   STATUS[822].EXT.AckRequired := FALSE;
   STATUS[822].EXT.Maintanence := FALSE;
   STATUS[822].EXT.Operation := FALSE;
   STATUS[822].EXT.Forced := FALSE;
   STATUS[822].EXT.BIT29 := FALSE;
   STATUS[822].EXT.BIT30 := FALSE;
   STATUS[822].EXT.BIT31 := FALSE;
   STATUS[822].EXT.ModeBit1 := FALSE;
   STATUS[822].EXT.ModeBit2 := FALSE;
   STATUS[822].EXT.ModeBit3 := FALSE;
   STATUS[822].EXT.BIT19 := FALSE;
   STATUS[822].EXT.BIT20 := FALSE;
   STATUS[822].EXT.AlarmSuppressed := FALSE;
   STATUS[822].EXT.AlarmPresent := FALSE;
   STATUS[822].EXT.AlarmFailUnAck := FALSE;
   STATUS[822].Status := 0;
   STATUS[822].TimeStamp := 16#0000;
   STATUS[823].EXT.AlarmWarnUnAck := FALSE;
   STATUS[823].EXT.AckRequired := FALSE;
   STATUS[823].EXT.Maintanence := FALSE;
   STATUS[823].EXT.Operation := FALSE;
   STATUS[823].EXT.Forced := FALSE;
   STATUS[823].EXT.BIT29 := FALSE;
   STATUS[823].EXT.BIT30 := FALSE;
   STATUS[823].EXT.BIT31 := FALSE;
   STATUS[823].EXT.ModeBit1 := FALSE;
   STATUS[823].EXT.ModeBit2 := FALSE;
   STATUS[823].EXT.ModeBit3 := FALSE;
   STATUS[823].EXT.BIT19 := FALSE;
   STATUS[823].EXT.BIT20 := FALSE;
   STATUS[823].EXT.AlarmSuppressed := FALSE;
   STATUS[823].EXT.AlarmPresent := FALSE;
   STATUS[823].EXT.AlarmFailUnAck := FALSE;
   STATUS[823].Status := 0;
   STATUS[823].TimeStamp := 16#0000;
   STATUS[824].EXT.AlarmWarnUnAck := FALSE;
   STATUS[824].EXT.AckRequired := FALSE;
   STATUS[824].EXT.Maintanence := FALSE;
   STATUS[824].EXT.Operation := FALSE;
   STATUS[824].EXT.Forced := FALSE;
   STATUS[824].EXT.BIT29 := FALSE;
   STATUS[824].EXT.BIT30 := FALSE;
   STATUS[824].EXT.BIT31 := FALSE;
   STATUS[824].EXT.ModeBit1 := FALSE;
   STATUS[824].EXT.ModeBit2 := FALSE;
   STATUS[824].EXT.ModeBit3 := FALSE;
   STATUS[824].EXT.BIT19 := FALSE;
   STATUS[824].EXT.BIT20 := FALSE;
   STATUS[824].EXT.AlarmSuppressed := FALSE;
   STATUS[824].EXT.AlarmPresent := FALSE;
   STATUS[824].EXT.AlarmFailUnAck := FALSE;
   STATUS[824].Status := 0;
   STATUS[824].TimeStamp := 16#0000;
   STATUS[825].EXT.AlarmWarnUnAck := FALSE;
   STATUS[825].EXT.AckRequired := FALSE;
   STATUS[825].EXT.Maintanence := FALSE;
   STATUS[825].EXT.Operation := FALSE;
   STATUS[825].EXT.Forced := FALSE;
   STATUS[825].EXT.BIT29 := FALSE;
   STATUS[825].EXT.BIT30 := FALSE;
   STATUS[825].EXT.BIT31 := FALSE;
   STATUS[825].EXT.ModeBit1 := FALSE;
   STATUS[825].EXT.ModeBit2 := FALSE;
   STATUS[825].EXT.ModeBit3 := FALSE;
   STATUS[825].EXT.BIT19 := FALSE;
   STATUS[825].EXT.BIT20 := FALSE;
   STATUS[825].EXT.AlarmSuppressed := FALSE;
   STATUS[825].EXT.AlarmPresent := FALSE;
   STATUS[825].EXT.AlarmFailUnAck := FALSE;
   STATUS[825].Status := 0;
   STATUS[825].TimeStamp := 16#0000;
   STATUS[826].EXT.AlarmWarnUnAck := FALSE;
   STATUS[826].EXT.AckRequired := FALSE;
   STATUS[826].EXT.Maintanence := FALSE;
   STATUS[826].EXT.Operation := FALSE;
   STATUS[826].EXT.Forced := FALSE;
   STATUS[826].EXT.BIT29 := FALSE;
   STATUS[826].EXT.BIT30 := FALSE;
   STATUS[826].EXT.BIT31 := FALSE;
   STATUS[826].EXT.ModeBit1 := FALSE;
   STATUS[826].EXT.ModeBit2 := FALSE;
   STATUS[826].EXT.ModeBit3 := FALSE;
   STATUS[826].EXT.BIT19 := FALSE;
   STATUS[826].EXT.BIT20 := FALSE;
   STATUS[826].EXT.AlarmSuppressed := FALSE;
   STATUS[826].EXT.AlarmPresent := FALSE;
   STATUS[826].EXT.AlarmFailUnAck := FALSE;
   STATUS[826].Status := 0;
   STATUS[826].TimeStamp := 16#0000;
   STATUS[827].EXT.AlarmWarnUnAck := FALSE;
   STATUS[827].EXT.AckRequired := FALSE;
   STATUS[827].EXT.Maintanence := FALSE;
   STATUS[827].EXT.Operation := FALSE;
   STATUS[827].EXT.Forced := FALSE;
   STATUS[827].EXT.BIT29 := FALSE;
   STATUS[827].EXT.BIT30 := FALSE;
   STATUS[827].EXT.BIT31 := FALSE;
   STATUS[827].EXT.ModeBit1 := FALSE;
   STATUS[827].EXT.ModeBit2 := FALSE;
   STATUS[827].EXT.ModeBit3 := FALSE;
   STATUS[827].EXT.BIT19 := FALSE;
   STATUS[827].EXT.BIT20 := FALSE;
   STATUS[827].EXT.AlarmSuppressed := FALSE;
   STATUS[827].EXT.AlarmPresent := FALSE;
   STATUS[827].EXT.AlarmFailUnAck := FALSE;
   STATUS[827].Status := 0;
   STATUS[827].TimeStamp := 16#0000;
   STATUS[828].EXT.AlarmWarnUnAck := FALSE;
   STATUS[828].EXT.AckRequired := FALSE;
   STATUS[828].EXT.Maintanence := FALSE;
   STATUS[828].EXT.Operation := FALSE;
   STATUS[828].EXT.Forced := FALSE;
   STATUS[828].EXT.BIT29 := FALSE;
   STATUS[828].EXT.BIT30 := FALSE;
   STATUS[828].EXT.BIT31 := FALSE;
   STATUS[828].EXT.ModeBit1 := FALSE;
   STATUS[828].EXT.ModeBit2 := FALSE;
   STATUS[828].EXT.ModeBit3 := FALSE;
   STATUS[828].EXT.BIT19 := FALSE;
   STATUS[828].EXT.BIT20 := FALSE;
   STATUS[828].EXT.AlarmSuppressed := FALSE;
   STATUS[828].EXT.AlarmPresent := FALSE;
   STATUS[828].EXT.AlarmFailUnAck := FALSE;
   STATUS[828].Status := 0;
   STATUS[828].TimeStamp := 16#0000;
   STATUS[829].EXT.AlarmWarnUnAck := FALSE;
   STATUS[829].EXT.AckRequired := FALSE;
   STATUS[829].EXT.Maintanence := FALSE;
   STATUS[829].EXT.Operation := FALSE;
   STATUS[829].EXT.Forced := FALSE;
   STATUS[829].EXT.BIT29 := FALSE;
   STATUS[829].EXT.BIT30 := FALSE;
   STATUS[829].EXT.BIT31 := FALSE;
   STATUS[829].EXT.ModeBit1 := FALSE;
   STATUS[829].EXT.ModeBit2 := FALSE;
   STATUS[829].EXT.ModeBit3 := FALSE;
   STATUS[829].EXT.BIT19 := FALSE;
   STATUS[829].EXT.BIT20 := FALSE;
   STATUS[829].EXT.AlarmSuppressed := FALSE;
   STATUS[829].EXT.AlarmPresent := FALSE;
   STATUS[829].EXT.AlarmFailUnAck := FALSE;
   STATUS[829].Status := 0;
   STATUS[829].TimeStamp := 16#0000;
   STATUS[830].EXT.AlarmWarnUnAck := FALSE;
   STATUS[830].EXT.AckRequired := FALSE;
   STATUS[830].EXT.Maintanence := FALSE;
   STATUS[830].EXT.Operation := FALSE;
   STATUS[830].EXT.Forced := FALSE;
   STATUS[830].EXT.BIT29 := FALSE;
   STATUS[830].EXT.BIT30 := FALSE;
   STATUS[830].EXT.BIT31 := FALSE;
   STATUS[830].EXT.ModeBit1 := FALSE;
   STATUS[830].EXT.ModeBit2 := FALSE;
   STATUS[830].EXT.ModeBit3 := FALSE;
   STATUS[830].EXT.BIT19 := FALSE;
   STATUS[830].EXT.BIT20 := FALSE;
   STATUS[830].EXT.AlarmSuppressed := FALSE;
   STATUS[830].EXT.AlarmPresent := FALSE;
   STATUS[830].EXT.AlarmFailUnAck := FALSE;
   STATUS[830].Status := 0;
   STATUS[830].TimeStamp := 16#0000;
   STATUS[831].EXT.AlarmWarnUnAck := FALSE;
   STATUS[831].EXT.AckRequired := FALSE;
   STATUS[831].EXT.Maintanence := FALSE;
   STATUS[831].EXT.Operation := FALSE;
   STATUS[831].EXT.Forced := FALSE;
   STATUS[831].EXT.BIT29 := FALSE;
   STATUS[831].EXT.BIT30 := FALSE;
   STATUS[831].EXT.BIT31 := FALSE;
   STATUS[831].EXT.ModeBit1 := FALSE;
   STATUS[831].EXT.ModeBit2 := FALSE;
   STATUS[831].EXT.ModeBit3 := FALSE;
   STATUS[831].EXT.BIT19 := FALSE;
   STATUS[831].EXT.BIT20 := FALSE;
   STATUS[831].EXT.AlarmSuppressed := FALSE;
   STATUS[831].EXT.AlarmPresent := FALSE;
   STATUS[831].EXT.AlarmFailUnAck := FALSE;
   STATUS[831].Status := 0;
   STATUS[831].TimeStamp := 16#0000;
   STATUS[832].EXT.AlarmWarnUnAck := FALSE;
   STATUS[832].EXT.AckRequired := FALSE;
   STATUS[832].EXT.Maintanence := FALSE;
   STATUS[832].EXT.Operation := FALSE;
   STATUS[832].EXT.Forced := FALSE;
   STATUS[832].EXT.BIT29 := FALSE;
   STATUS[832].EXT.BIT30 := FALSE;
   STATUS[832].EXT.BIT31 := FALSE;
   STATUS[832].EXT.ModeBit1 := FALSE;
   STATUS[832].EXT.ModeBit2 := FALSE;
   STATUS[832].EXT.ModeBit3 := FALSE;
   STATUS[832].EXT.BIT19 := FALSE;
   STATUS[832].EXT.BIT20 := FALSE;
   STATUS[832].EXT.AlarmSuppressed := FALSE;
   STATUS[832].EXT.AlarmPresent := FALSE;
   STATUS[832].EXT.AlarmFailUnAck := FALSE;
   STATUS[832].Status := 0;
   STATUS[832].TimeStamp := 16#0000;
   STATUS[833].EXT.AlarmWarnUnAck := FALSE;
   STATUS[833].EXT.AckRequired := FALSE;
   STATUS[833].EXT.Maintanence := FALSE;
   STATUS[833].EXT.Operation := FALSE;
   STATUS[833].EXT.Forced := FALSE;
   STATUS[833].EXT.BIT29 := FALSE;
   STATUS[833].EXT.BIT30 := FALSE;
   STATUS[833].EXT.BIT31 := FALSE;
   STATUS[833].EXT.ModeBit1 := FALSE;
   STATUS[833].EXT.ModeBit2 := FALSE;
   STATUS[833].EXT.ModeBit3 := FALSE;
   STATUS[833].EXT.BIT19 := FALSE;
   STATUS[833].EXT.BIT20 := FALSE;
   STATUS[833].EXT.AlarmSuppressed := FALSE;
   STATUS[833].EXT.AlarmPresent := FALSE;
   STATUS[833].EXT.AlarmFailUnAck := FALSE;
   STATUS[833].Status := 0;
   STATUS[833].TimeStamp := 16#0000;
   STATUS[834].EXT.AlarmWarnUnAck := FALSE;
   STATUS[834].EXT.AckRequired := FALSE;
   STATUS[834].EXT.Maintanence := FALSE;
   STATUS[834].EXT.Operation := FALSE;
   STATUS[834].EXT.Forced := FALSE;
   STATUS[834].EXT.BIT29 := FALSE;
   STATUS[834].EXT.BIT30 := FALSE;
   STATUS[834].EXT.BIT31 := FALSE;
   STATUS[834].EXT.ModeBit1 := FALSE;
   STATUS[834].EXT.ModeBit2 := FALSE;
   STATUS[834].EXT.ModeBit3 := FALSE;
   STATUS[834].EXT.BIT19 := FALSE;
   STATUS[834].EXT.BIT20 := FALSE;
   STATUS[834].EXT.AlarmSuppressed := FALSE;
   STATUS[834].EXT.AlarmPresent := FALSE;
   STATUS[834].EXT.AlarmFailUnAck := FALSE;
   STATUS[834].Status := 0;
   STATUS[834].TimeStamp := 16#0000;
   STATUS[835].EXT.AlarmWarnUnAck := FALSE;
   STATUS[835].EXT.AckRequired := FALSE;
   STATUS[835].EXT.Maintanence := FALSE;
   STATUS[835].EXT.Operation := FALSE;
   STATUS[835].EXT.Forced := FALSE;
   STATUS[835].EXT.BIT29 := FALSE;
   STATUS[835].EXT.BIT30 := FALSE;
   STATUS[835].EXT.BIT31 := FALSE;
   STATUS[835].EXT.ModeBit1 := FALSE;
   STATUS[835].EXT.ModeBit2 := FALSE;
   STATUS[835].EXT.ModeBit3 := FALSE;
   STATUS[835].EXT.BIT19 := FALSE;
   STATUS[835].EXT.BIT20 := FALSE;
   STATUS[835].EXT.AlarmSuppressed := FALSE;
   STATUS[835].EXT.AlarmPresent := FALSE;
   STATUS[835].EXT.AlarmFailUnAck := FALSE;
   STATUS[835].Status := 0;
   STATUS[835].TimeStamp := 16#0000;
   STATUS[836].EXT.AlarmWarnUnAck := FALSE;
   STATUS[836].EXT.AckRequired := FALSE;
   STATUS[836].EXT.Maintanence := FALSE;
   STATUS[836].EXT.Operation := FALSE;
   STATUS[836].EXT.Forced := FALSE;
   STATUS[836].EXT.BIT29 := FALSE;
   STATUS[836].EXT.BIT30 := FALSE;
   STATUS[836].EXT.BIT31 := FALSE;
   STATUS[836].EXT.ModeBit1 := FALSE;
   STATUS[836].EXT.ModeBit2 := FALSE;
   STATUS[836].EXT.ModeBit3 := FALSE;
   STATUS[836].EXT.BIT19 := FALSE;
   STATUS[836].EXT.BIT20 := FALSE;
   STATUS[836].EXT.AlarmSuppressed := FALSE;
   STATUS[836].EXT.AlarmPresent := FALSE;
   STATUS[836].EXT.AlarmFailUnAck := FALSE;
   STATUS[836].Status := 0;
   STATUS[836].TimeStamp := 16#0000;
   STATUS[837].EXT.AlarmWarnUnAck := FALSE;
   STATUS[837].EXT.AckRequired := FALSE;
   STATUS[837].EXT.Maintanence := FALSE;
   STATUS[837].EXT.Operation := FALSE;
   STATUS[837].EXT.Forced := FALSE;
   STATUS[837].EXT.BIT29 := FALSE;
   STATUS[837].EXT.BIT30 := FALSE;
   STATUS[837].EXT.BIT31 := FALSE;
   STATUS[837].EXT.ModeBit1 := FALSE;
   STATUS[837].EXT.ModeBit2 := FALSE;
   STATUS[837].EXT.ModeBit3 := FALSE;
   STATUS[837].EXT.BIT19 := FALSE;
   STATUS[837].EXT.BIT20 := FALSE;
   STATUS[837].EXT.AlarmSuppressed := FALSE;
   STATUS[837].EXT.AlarmPresent := FALSE;
   STATUS[837].EXT.AlarmFailUnAck := FALSE;
   STATUS[837].Status := 0;
   STATUS[837].TimeStamp := 16#0000;
   STATUS[838].EXT.AlarmWarnUnAck := FALSE;
   STATUS[838].EXT.AckRequired := FALSE;
   STATUS[838].EXT.Maintanence := FALSE;
   STATUS[838].EXT.Operation := FALSE;
   STATUS[838].EXT.Forced := FALSE;
   STATUS[838].EXT.BIT29 := FALSE;
   STATUS[838].EXT.BIT30 := FALSE;
   STATUS[838].EXT.BIT31 := FALSE;
   STATUS[838].EXT.ModeBit1 := FALSE;
   STATUS[838].EXT.ModeBit2 := FALSE;
   STATUS[838].EXT.ModeBit3 := FALSE;
   STATUS[838].EXT.BIT19 := FALSE;
   STATUS[838].EXT.BIT20 := FALSE;
   STATUS[838].EXT.AlarmSuppressed := FALSE;
   STATUS[838].EXT.AlarmPresent := FALSE;
   STATUS[838].EXT.AlarmFailUnAck := FALSE;
   STATUS[838].Status := 0;
   STATUS[838].TimeStamp := 16#0000;
   STATUS[839].EXT.AlarmWarnUnAck := FALSE;
   STATUS[839].EXT.AckRequired := FALSE;
   STATUS[839].EXT.Maintanence := FALSE;
   STATUS[839].EXT.Operation := FALSE;
   STATUS[839].EXT.Forced := FALSE;
   STATUS[839].EXT.BIT29 := FALSE;
   STATUS[839].EXT.BIT30 := FALSE;
   STATUS[839].EXT.BIT31 := FALSE;
   STATUS[839].EXT.ModeBit1 := FALSE;
   STATUS[839].EXT.ModeBit2 := FALSE;
   STATUS[839].EXT.ModeBit3 := FALSE;
   STATUS[839].EXT.BIT19 := FALSE;
   STATUS[839].EXT.BIT20 := FALSE;
   STATUS[839].EXT.AlarmSuppressed := FALSE;
   STATUS[839].EXT.AlarmPresent := FALSE;
   STATUS[839].EXT.AlarmFailUnAck := FALSE;
   STATUS[839].Status := 0;
   STATUS[839].TimeStamp := 16#0000;
   STATUS[840].EXT.AlarmWarnUnAck := FALSE;
   STATUS[840].EXT.AckRequired := FALSE;
   STATUS[840].EXT.Maintanence := FALSE;
   STATUS[840].EXT.Operation := FALSE;
   STATUS[840].EXT.Forced := FALSE;
   STATUS[840].EXT.BIT29 := FALSE;
   STATUS[840].EXT.BIT30 := FALSE;
   STATUS[840].EXT.BIT31 := FALSE;
   STATUS[840].EXT.ModeBit1 := FALSE;
   STATUS[840].EXT.ModeBit2 := FALSE;
   STATUS[840].EXT.ModeBit3 := FALSE;
   STATUS[840].EXT.BIT19 := FALSE;
   STATUS[840].EXT.BIT20 := FALSE;
   STATUS[840].EXT.AlarmSuppressed := FALSE;
   STATUS[840].EXT.AlarmPresent := FALSE;
   STATUS[840].EXT.AlarmFailUnAck := FALSE;
   STATUS[840].Status := 0;
   STATUS[840].TimeStamp := 16#0000;
   STATUS[841].EXT.AlarmWarnUnAck := FALSE;
   STATUS[841].EXT.AckRequired := FALSE;
   STATUS[841].EXT.Maintanence := FALSE;
   STATUS[841].EXT.Operation := FALSE;
   STATUS[841].EXT.Forced := FALSE;
   STATUS[841].EXT.BIT29 := FALSE;
   STATUS[841].EXT.BIT30 := FALSE;
   STATUS[841].EXT.BIT31 := FALSE;
   STATUS[841].EXT.ModeBit1 := FALSE;
   STATUS[841].EXT.ModeBit2 := FALSE;
   STATUS[841].EXT.ModeBit3 := FALSE;
   STATUS[841].EXT.BIT19 := FALSE;
   STATUS[841].EXT.BIT20 := FALSE;
   STATUS[841].EXT.AlarmSuppressed := FALSE;
   STATUS[841].EXT.AlarmPresent := FALSE;
   STATUS[841].EXT.AlarmFailUnAck := FALSE;
   STATUS[841].Status := 0;
   STATUS[841].TimeStamp := 16#0000;
   STATUS[842].EXT.AlarmWarnUnAck := FALSE;
   STATUS[842].EXT.AckRequired := FALSE;
   STATUS[842].EXT.Maintanence := FALSE;
   STATUS[842].EXT.Operation := FALSE;
   STATUS[842].EXT.Forced := FALSE;
   STATUS[842].EXT.BIT29 := FALSE;
   STATUS[842].EXT.BIT30 := FALSE;
   STATUS[842].EXT.BIT31 := FALSE;
   STATUS[842].EXT.ModeBit1 := FALSE;
   STATUS[842].EXT.ModeBit2 := FALSE;
   STATUS[842].EXT.ModeBit3 := FALSE;
   STATUS[842].EXT.BIT19 := FALSE;
   STATUS[842].EXT.BIT20 := FALSE;
   STATUS[842].EXT.AlarmSuppressed := FALSE;
   STATUS[842].EXT.AlarmPresent := FALSE;
   STATUS[842].EXT.AlarmFailUnAck := FALSE;
   STATUS[842].Status := 0;
   STATUS[842].TimeStamp := 16#0000;
   STATUS[843].EXT.AlarmWarnUnAck := FALSE;
   STATUS[843].EXT.AckRequired := FALSE;
   STATUS[843].EXT.Maintanence := FALSE;
   STATUS[843].EXT.Operation := FALSE;
   STATUS[843].EXT.Forced := FALSE;
   STATUS[843].EXT.BIT29 := FALSE;
   STATUS[843].EXT.BIT30 := FALSE;
   STATUS[843].EXT.BIT31 := FALSE;
   STATUS[843].EXT.ModeBit1 := FALSE;
   STATUS[843].EXT.ModeBit2 := FALSE;
   STATUS[843].EXT.ModeBit3 := FALSE;
   STATUS[843].EXT.BIT19 := FALSE;
   STATUS[843].EXT.BIT20 := FALSE;
   STATUS[843].EXT.AlarmSuppressed := FALSE;
   STATUS[843].EXT.AlarmPresent := FALSE;
   STATUS[843].EXT.AlarmFailUnAck := FALSE;
   STATUS[843].Status := 0;
   STATUS[843].TimeStamp := 16#0000;
   STATUS[844].EXT.AlarmWarnUnAck := FALSE;
   STATUS[844].EXT.AckRequired := FALSE;
   STATUS[844].EXT.Maintanence := FALSE;
   STATUS[844].EXT.Operation := FALSE;
   STATUS[844].EXT.Forced := FALSE;
   STATUS[844].EXT.BIT29 := FALSE;
   STATUS[844].EXT.BIT30 := FALSE;
   STATUS[844].EXT.BIT31 := FALSE;
   STATUS[844].EXT.ModeBit1 := FALSE;
   STATUS[844].EXT.ModeBit2 := FALSE;
   STATUS[844].EXT.ModeBit3 := FALSE;
   STATUS[844].EXT.BIT19 := FALSE;
   STATUS[844].EXT.BIT20 := FALSE;
   STATUS[844].EXT.AlarmSuppressed := FALSE;
   STATUS[844].EXT.AlarmPresent := FALSE;
   STATUS[844].EXT.AlarmFailUnAck := FALSE;
   STATUS[844].Status := 0;
   STATUS[844].TimeStamp := 16#0000;
   STATUS[845].EXT.AlarmWarnUnAck := FALSE;
   STATUS[845].EXT.AckRequired := FALSE;
   STATUS[845].EXT.Maintanence := FALSE;
   STATUS[845].EXT.Operation := FALSE;
   STATUS[845].EXT.Forced := FALSE;
   STATUS[845].EXT.BIT29 := FALSE;
   STATUS[845].EXT.BIT30 := FALSE;
   STATUS[845].EXT.BIT31 := FALSE;
   STATUS[845].EXT.ModeBit1 := FALSE;
   STATUS[845].EXT.ModeBit2 := FALSE;
   STATUS[845].EXT.ModeBit3 := FALSE;
   STATUS[845].EXT.BIT19 := FALSE;
   STATUS[845].EXT.BIT20 := FALSE;
   STATUS[845].EXT.AlarmSuppressed := FALSE;
   STATUS[845].EXT.AlarmPresent := FALSE;
   STATUS[845].EXT.AlarmFailUnAck := FALSE;
   STATUS[845].Status := 0;
   STATUS[845].TimeStamp := 16#0000;
   STATUS[846].EXT.AlarmWarnUnAck := FALSE;
   STATUS[846].EXT.AckRequired := FALSE;
   STATUS[846].EXT.Maintanence := FALSE;
   STATUS[846].EXT.Operation := FALSE;
   STATUS[846].EXT.Forced := FALSE;
   STATUS[846].EXT.BIT29 := FALSE;
   STATUS[846].EXT.BIT30 := FALSE;
   STATUS[846].EXT.BIT31 := FALSE;
   STATUS[846].EXT.ModeBit1 := FALSE;
   STATUS[846].EXT.ModeBit2 := FALSE;
   STATUS[846].EXT.ModeBit3 := FALSE;
   STATUS[846].EXT.BIT19 := FALSE;
   STATUS[846].EXT.BIT20 := FALSE;
   STATUS[846].EXT.AlarmSuppressed := FALSE;
   STATUS[846].EXT.AlarmPresent := FALSE;
   STATUS[846].EXT.AlarmFailUnAck := FALSE;
   STATUS[846].Status := 0;
   STATUS[846].TimeStamp := 16#0000;
   STATUS[847].EXT.AlarmWarnUnAck := FALSE;
   STATUS[847].EXT.AckRequired := FALSE;
   STATUS[847].EXT.Maintanence := FALSE;
   STATUS[847].EXT.Operation := FALSE;
   STATUS[847].EXT.Forced := FALSE;
   STATUS[847].EXT.BIT29 := FALSE;
   STATUS[847].EXT.BIT30 := FALSE;
   STATUS[847].EXT.BIT31 := FALSE;
   STATUS[847].EXT.ModeBit1 := FALSE;
   STATUS[847].EXT.ModeBit2 := FALSE;
   STATUS[847].EXT.ModeBit3 := FALSE;
   STATUS[847].EXT.BIT19 := FALSE;
   STATUS[847].EXT.BIT20 := FALSE;
   STATUS[847].EXT.AlarmSuppressed := FALSE;
   STATUS[847].EXT.AlarmPresent := FALSE;
   STATUS[847].EXT.AlarmFailUnAck := FALSE;
   STATUS[847].Status := 0;
   STATUS[847].TimeStamp := 16#0000;
   STATUS[848].EXT.AlarmWarnUnAck := FALSE;
   STATUS[848].EXT.AckRequired := FALSE;
   STATUS[848].EXT.Maintanence := FALSE;
   STATUS[848].EXT.Operation := FALSE;
   STATUS[848].EXT.Forced := FALSE;
   STATUS[848].EXT.BIT29 := FALSE;
   STATUS[848].EXT.BIT30 := FALSE;
   STATUS[848].EXT.BIT31 := FALSE;
   STATUS[848].EXT.ModeBit1 := FALSE;
   STATUS[848].EXT.ModeBit2 := FALSE;
   STATUS[848].EXT.ModeBit3 := FALSE;
   STATUS[848].EXT.BIT19 := FALSE;
   STATUS[848].EXT.BIT20 := FALSE;
   STATUS[848].EXT.AlarmSuppressed := FALSE;
   STATUS[848].EXT.AlarmPresent := FALSE;
   STATUS[848].EXT.AlarmFailUnAck := FALSE;
   STATUS[848].Status := 0;
   STATUS[848].TimeStamp := 16#0000;
   STATUS[849].EXT.AlarmWarnUnAck := FALSE;
   STATUS[849].EXT.AckRequired := FALSE;
   STATUS[849].EXT.Maintanence := FALSE;
   STATUS[849].EXT.Operation := FALSE;
   STATUS[849].EXT.Forced := FALSE;
   STATUS[849].EXT.BIT29 := FALSE;
   STATUS[849].EXT.BIT30 := FALSE;
   STATUS[849].EXT.BIT31 := FALSE;
   STATUS[849].EXT.ModeBit1 := FALSE;
   STATUS[849].EXT.ModeBit2 := FALSE;
   STATUS[849].EXT.ModeBit3 := FALSE;
   STATUS[849].EXT.BIT19 := FALSE;
   STATUS[849].EXT.BIT20 := FALSE;
   STATUS[849].EXT.AlarmSuppressed := FALSE;
   STATUS[849].EXT.AlarmPresent := FALSE;
   STATUS[849].EXT.AlarmFailUnAck := FALSE;
   STATUS[849].Status := 0;
   STATUS[849].TimeStamp := 16#0000;
   STATUS[850].EXT.AlarmWarnUnAck := FALSE;
   STATUS[850].EXT.AckRequired := FALSE;
   STATUS[850].EXT.Maintanence := FALSE;
   STATUS[850].EXT.Operation := FALSE;
   STATUS[850].EXT.Forced := FALSE;
   STATUS[850].EXT.BIT29 := FALSE;
   STATUS[850].EXT.BIT30 := FALSE;
   STATUS[850].EXT.BIT31 := FALSE;
   STATUS[850].EXT.ModeBit1 := FALSE;
   STATUS[850].EXT.ModeBit2 := FALSE;
   STATUS[850].EXT.ModeBit3 := FALSE;
   STATUS[850].EXT.BIT19 := FALSE;
   STATUS[850].EXT.BIT20 := FALSE;
   STATUS[850].EXT.AlarmSuppressed := FALSE;
   STATUS[850].EXT.AlarmPresent := FALSE;
   STATUS[850].EXT.AlarmFailUnAck := FALSE;
   STATUS[850].Status := 0;
   STATUS[850].TimeStamp := 16#0000;
   STATUS[851].EXT.AlarmWarnUnAck := FALSE;
   STATUS[851].EXT.AckRequired := FALSE;
   STATUS[851].EXT.Maintanence := FALSE;
   STATUS[851].EXT.Operation := FALSE;
   STATUS[851].EXT.Forced := FALSE;
   STATUS[851].EXT.BIT29 := FALSE;
   STATUS[851].EXT.BIT30 := FALSE;
   STATUS[851].EXT.BIT31 := FALSE;
   STATUS[851].EXT.ModeBit1 := FALSE;
   STATUS[851].EXT.ModeBit2 := FALSE;
   STATUS[851].EXT.ModeBit3 := FALSE;
   STATUS[851].EXT.BIT19 := FALSE;
   STATUS[851].EXT.BIT20 := FALSE;
   STATUS[851].EXT.AlarmSuppressed := FALSE;
   STATUS[851].EXT.AlarmPresent := FALSE;
   STATUS[851].EXT.AlarmFailUnAck := FALSE;
   STATUS[851].Status := 0;
   STATUS[851].TimeStamp := 16#0000;
   STATUS[852].EXT.AlarmWarnUnAck := FALSE;
   STATUS[852].EXT.AckRequired := FALSE;
   STATUS[852].EXT.Maintanence := FALSE;
   STATUS[852].EXT.Operation := FALSE;
   STATUS[852].EXT.Forced := FALSE;
   STATUS[852].EXT.BIT29 := FALSE;
   STATUS[852].EXT.BIT30 := FALSE;
   STATUS[852].EXT.BIT31 := FALSE;
   STATUS[852].EXT.ModeBit1 := FALSE;
   STATUS[852].EXT.ModeBit2 := FALSE;
   STATUS[852].EXT.ModeBit3 := FALSE;
   STATUS[852].EXT.BIT19 := FALSE;
   STATUS[852].EXT.BIT20 := FALSE;
   STATUS[852].EXT.AlarmSuppressed := FALSE;
   STATUS[852].EXT.AlarmPresent := FALSE;
   STATUS[852].EXT.AlarmFailUnAck := FALSE;
   STATUS[852].Status := 0;
   STATUS[852].TimeStamp := 16#0000;
   STATUS[853].EXT.AlarmWarnUnAck := FALSE;
   STATUS[853].EXT.AckRequired := FALSE;
   STATUS[853].EXT.Maintanence := FALSE;
   STATUS[853].EXT.Operation := FALSE;
   STATUS[853].EXT.Forced := FALSE;
   STATUS[853].EXT.BIT29 := FALSE;
   STATUS[853].EXT.BIT30 := FALSE;
   STATUS[853].EXT.BIT31 := FALSE;
   STATUS[853].EXT.ModeBit1 := FALSE;
   STATUS[853].EXT.ModeBit2 := FALSE;
   STATUS[853].EXT.ModeBit3 := FALSE;
   STATUS[853].EXT.BIT19 := FALSE;
   STATUS[853].EXT.BIT20 := FALSE;
   STATUS[853].EXT.AlarmSuppressed := FALSE;
   STATUS[853].EXT.AlarmPresent := FALSE;
   STATUS[853].EXT.AlarmFailUnAck := FALSE;
   STATUS[853].Status := 0;
   STATUS[853].TimeStamp := 16#0000;
   STATUS[854].EXT.AlarmWarnUnAck := FALSE;
   STATUS[854].EXT.AckRequired := FALSE;
   STATUS[854].EXT.Maintanence := FALSE;
   STATUS[854].EXT.Operation := FALSE;
   STATUS[854].EXT.Forced := FALSE;
   STATUS[854].EXT.BIT29 := FALSE;
   STATUS[854].EXT.BIT30 := FALSE;
   STATUS[854].EXT.BIT31 := FALSE;
   STATUS[854].EXT.ModeBit1 := FALSE;
   STATUS[854].EXT.ModeBit2 := FALSE;
   STATUS[854].EXT.ModeBit3 := FALSE;
   STATUS[854].EXT.BIT19 := FALSE;
   STATUS[854].EXT.BIT20 := FALSE;
   STATUS[854].EXT.AlarmSuppressed := FALSE;
   STATUS[854].EXT.AlarmPresent := FALSE;
   STATUS[854].EXT.AlarmFailUnAck := FALSE;
   STATUS[854].Status := 0;
   STATUS[854].TimeStamp := 16#0000;
   STATUS[855].EXT.AlarmWarnUnAck := FALSE;
   STATUS[855].EXT.AckRequired := FALSE;
   STATUS[855].EXT.Maintanence := FALSE;
   STATUS[855].EXT.Operation := FALSE;
   STATUS[855].EXT.Forced := FALSE;
   STATUS[855].EXT.BIT29 := FALSE;
   STATUS[855].EXT.BIT30 := FALSE;
   STATUS[855].EXT.BIT31 := FALSE;
   STATUS[855].EXT.ModeBit1 := FALSE;
   STATUS[855].EXT.ModeBit2 := FALSE;
   STATUS[855].EXT.ModeBit3 := FALSE;
   STATUS[855].EXT.BIT19 := FALSE;
   STATUS[855].EXT.BIT20 := FALSE;
   STATUS[855].EXT.AlarmSuppressed := FALSE;
   STATUS[855].EXT.AlarmPresent := FALSE;
   STATUS[855].EXT.AlarmFailUnAck := FALSE;
   STATUS[855].Status := 0;
   STATUS[855].TimeStamp := 16#0000;
   STATUS[856].EXT.AlarmWarnUnAck := FALSE;
   STATUS[856].EXT.AckRequired := FALSE;
   STATUS[856].EXT.Maintanence := FALSE;
   STATUS[856].EXT.Operation := FALSE;
   STATUS[856].EXT.Forced := FALSE;
   STATUS[856].EXT.BIT29 := FALSE;
   STATUS[856].EXT.BIT30 := FALSE;
   STATUS[856].EXT.BIT31 := FALSE;
   STATUS[856].EXT.ModeBit1 := FALSE;
   STATUS[856].EXT.ModeBit2 := FALSE;
   STATUS[856].EXT.ModeBit3 := FALSE;
   STATUS[856].EXT.BIT19 := FALSE;
   STATUS[856].EXT.BIT20 := FALSE;
   STATUS[856].EXT.AlarmSuppressed := FALSE;
   STATUS[856].EXT.AlarmPresent := FALSE;
   STATUS[856].EXT.AlarmFailUnAck := FALSE;
   STATUS[856].Status := 0;
   STATUS[856].TimeStamp := 16#0000;
   STATUS[857].EXT.AlarmWarnUnAck := FALSE;
   STATUS[857].EXT.AckRequired := FALSE;
   STATUS[857].EXT.Maintanence := FALSE;
   STATUS[857].EXT.Operation := FALSE;
   STATUS[857].EXT.Forced := FALSE;
   STATUS[857].EXT.BIT29 := FALSE;
   STATUS[857].EXT.BIT30 := FALSE;
   STATUS[857].EXT.BIT31 := FALSE;
   STATUS[857].EXT.ModeBit1 := FALSE;
   STATUS[857].EXT.ModeBit2 := FALSE;
   STATUS[857].EXT.ModeBit3 := FALSE;
   STATUS[857].EXT.BIT19 := FALSE;
   STATUS[857].EXT.BIT20 := FALSE;
   STATUS[857].EXT.AlarmSuppressed := FALSE;
   STATUS[857].EXT.AlarmPresent := FALSE;
   STATUS[857].EXT.AlarmFailUnAck := FALSE;
   STATUS[857].Status := 0;
   STATUS[857].TimeStamp := 16#0000;
   STATUS[858].EXT.AlarmWarnUnAck := FALSE;
   STATUS[858].EXT.AckRequired := FALSE;
   STATUS[858].EXT.Maintanence := FALSE;
   STATUS[858].EXT.Operation := FALSE;
   STATUS[858].EXT.Forced := FALSE;
   STATUS[858].EXT.BIT29 := FALSE;
   STATUS[858].EXT.BIT30 := FALSE;
   STATUS[858].EXT.BIT31 := FALSE;
   STATUS[858].EXT.ModeBit1 := FALSE;
   STATUS[858].EXT.ModeBit2 := FALSE;
   STATUS[858].EXT.ModeBit3 := FALSE;
   STATUS[858].EXT.BIT19 := FALSE;
   STATUS[858].EXT.BIT20 := FALSE;
   STATUS[858].EXT.AlarmSuppressed := FALSE;
   STATUS[858].EXT.AlarmPresent := FALSE;
   STATUS[858].EXT.AlarmFailUnAck := FALSE;
   STATUS[858].Status := 0;
   STATUS[858].TimeStamp := 16#0000;
   STATUS[859].EXT.AlarmWarnUnAck := FALSE;
   STATUS[859].EXT.AckRequired := FALSE;
   STATUS[859].EXT.Maintanence := FALSE;
   STATUS[859].EXT.Operation := FALSE;
   STATUS[859].EXT.Forced := FALSE;
   STATUS[859].EXT.BIT29 := FALSE;
   STATUS[859].EXT.BIT30 := FALSE;
   STATUS[859].EXT.BIT31 := FALSE;
   STATUS[859].EXT.ModeBit1 := FALSE;
   STATUS[859].EXT.ModeBit2 := FALSE;
   STATUS[859].EXT.ModeBit3 := FALSE;
   STATUS[859].EXT.BIT19 := FALSE;
   STATUS[859].EXT.BIT20 := FALSE;
   STATUS[859].EXT.AlarmSuppressed := FALSE;
   STATUS[859].EXT.AlarmPresent := FALSE;
   STATUS[859].EXT.AlarmFailUnAck := FALSE;
   STATUS[859].Status := 0;
   STATUS[859].TimeStamp := 16#0000;
   STATUS[860].EXT.AlarmWarnUnAck := FALSE;
   STATUS[860].EXT.AckRequired := FALSE;
   STATUS[860].EXT.Maintanence := FALSE;
   STATUS[860].EXT.Operation := FALSE;
   STATUS[860].EXT.Forced := FALSE;
   STATUS[860].EXT.BIT29 := FALSE;
   STATUS[860].EXT.BIT30 := FALSE;
   STATUS[860].EXT.BIT31 := FALSE;
   STATUS[860].EXT.ModeBit1 := FALSE;
   STATUS[860].EXT.ModeBit2 := FALSE;
   STATUS[860].EXT.ModeBit3 := FALSE;
   STATUS[860].EXT.BIT19 := FALSE;
   STATUS[860].EXT.BIT20 := FALSE;
   STATUS[860].EXT.AlarmSuppressed := FALSE;
   STATUS[860].EXT.AlarmPresent := FALSE;
   STATUS[860].EXT.AlarmFailUnAck := FALSE;
   STATUS[860].Status := 0;
   STATUS[860].TimeStamp := 16#0000;
   STATUS[861].EXT.AlarmWarnUnAck := FALSE;
   STATUS[861].EXT.AckRequired := FALSE;
   STATUS[861].EXT.Maintanence := FALSE;
   STATUS[861].EXT.Operation := FALSE;
   STATUS[861].EXT.Forced := FALSE;
   STATUS[861].EXT.BIT29 := FALSE;
   STATUS[861].EXT.BIT30 := FALSE;
   STATUS[861].EXT.BIT31 := FALSE;
   STATUS[861].EXT.ModeBit1 := FALSE;
   STATUS[861].EXT.ModeBit2 := FALSE;
   STATUS[861].EXT.ModeBit3 := FALSE;
   STATUS[861].EXT.BIT19 := FALSE;
   STATUS[861].EXT.BIT20 := FALSE;
   STATUS[861].EXT.AlarmSuppressed := FALSE;
   STATUS[861].EXT.AlarmPresent := FALSE;
   STATUS[861].EXT.AlarmFailUnAck := FALSE;
   STATUS[861].Status := 0;
   STATUS[861].TimeStamp := 16#0000;
   STATUS[862].EXT.AlarmWarnUnAck := FALSE;
   STATUS[862].EXT.AckRequired := FALSE;
   STATUS[862].EXT.Maintanence := FALSE;
   STATUS[862].EXT.Operation := FALSE;
   STATUS[862].EXT.Forced := FALSE;
   STATUS[862].EXT.BIT29 := FALSE;
   STATUS[862].EXT.BIT30 := FALSE;
   STATUS[862].EXT.BIT31 := FALSE;
   STATUS[862].EXT.ModeBit1 := FALSE;
   STATUS[862].EXT.ModeBit2 := FALSE;
   STATUS[862].EXT.ModeBit3 := FALSE;
   STATUS[862].EXT.BIT19 := FALSE;
   STATUS[862].EXT.BIT20 := FALSE;
   STATUS[862].EXT.AlarmSuppressed := FALSE;
   STATUS[862].EXT.AlarmPresent := FALSE;
   STATUS[862].EXT.AlarmFailUnAck := FALSE;
   STATUS[862].Status := 0;
   STATUS[862].TimeStamp := 16#0000;
   STATUS[863].EXT.AlarmWarnUnAck := FALSE;
   STATUS[863].EXT.AckRequired := FALSE;
   STATUS[863].EXT.Maintanence := FALSE;
   STATUS[863].EXT.Operation := FALSE;
   STATUS[863].EXT.Forced := FALSE;
   STATUS[863].EXT.BIT29 := FALSE;
   STATUS[863].EXT.BIT30 := FALSE;
   STATUS[863].EXT.BIT31 := FALSE;
   STATUS[863].EXT.ModeBit1 := FALSE;
   STATUS[863].EXT.ModeBit2 := FALSE;
   STATUS[863].EXT.ModeBit3 := FALSE;
   STATUS[863].EXT.BIT19 := FALSE;
   STATUS[863].EXT.BIT20 := FALSE;
   STATUS[863].EXT.AlarmSuppressed := FALSE;
   STATUS[863].EXT.AlarmPresent := FALSE;
   STATUS[863].EXT.AlarmFailUnAck := FALSE;
   STATUS[863].Status := 0;
   STATUS[863].TimeStamp := 16#0000;
   STATUS[864].EXT.AlarmWarnUnAck := FALSE;
   STATUS[864].EXT.AckRequired := FALSE;
   STATUS[864].EXT.Maintanence := FALSE;
   STATUS[864].EXT.Operation := FALSE;
   STATUS[864].EXT.Forced := FALSE;
   STATUS[864].EXT.BIT29 := FALSE;
   STATUS[864].EXT.BIT30 := FALSE;
   STATUS[864].EXT.BIT31 := FALSE;
   STATUS[864].EXT.ModeBit1 := FALSE;
   STATUS[864].EXT.ModeBit2 := FALSE;
   STATUS[864].EXT.ModeBit3 := FALSE;
   STATUS[864].EXT.BIT19 := FALSE;
   STATUS[864].EXT.BIT20 := FALSE;
   STATUS[864].EXT.AlarmSuppressed := FALSE;
   STATUS[864].EXT.AlarmPresent := FALSE;
   STATUS[864].EXT.AlarmFailUnAck := FALSE;
   STATUS[864].Status := 0;
   STATUS[864].TimeStamp := 16#0000;
   STATUS[865].EXT.AlarmWarnUnAck := FALSE;
   STATUS[865].EXT.AckRequired := FALSE;
   STATUS[865].EXT.Maintanence := FALSE;
   STATUS[865].EXT.Operation := FALSE;
   STATUS[865].EXT.Forced := FALSE;
   STATUS[865].EXT.BIT29 := FALSE;
   STATUS[865].EXT.BIT30 := FALSE;
   STATUS[865].EXT.BIT31 := FALSE;
   STATUS[865].EXT.ModeBit1 := FALSE;
   STATUS[865].EXT.ModeBit2 := FALSE;
   STATUS[865].EXT.ModeBit3 := FALSE;
   STATUS[865].EXT.BIT19 := FALSE;
   STATUS[865].EXT.BIT20 := FALSE;
   STATUS[865].EXT.AlarmSuppressed := FALSE;
   STATUS[865].EXT.AlarmPresent := FALSE;
   STATUS[865].EXT.AlarmFailUnAck := FALSE;
   STATUS[865].Status := 0;
   STATUS[865].TimeStamp := 16#0000;
   STATUS[866].EXT.AlarmWarnUnAck := FALSE;
   STATUS[866].EXT.AckRequired := FALSE;
   STATUS[866].EXT.Maintanence := FALSE;
   STATUS[866].EXT.Operation := FALSE;
   STATUS[866].EXT.Forced := FALSE;
   STATUS[866].EXT.BIT29 := FALSE;
   STATUS[866].EXT.BIT30 := FALSE;
   STATUS[866].EXT.BIT31 := FALSE;
   STATUS[866].EXT.ModeBit1 := FALSE;
   STATUS[866].EXT.ModeBit2 := FALSE;
   STATUS[866].EXT.ModeBit3 := FALSE;
   STATUS[866].EXT.BIT19 := FALSE;
   STATUS[866].EXT.BIT20 := FALSE;
   STATUS[866].EXT.AlarmSuppressed := FALSE;
   STATUS[866].EXT.AlarmPresent := FALSE;
   STATUS[866].EXT.AlarmFailUnAck := FALSE;
   STATUS[866].Status := 0;
   STATUS[866].TimeStamp := 16#0000;
   STATUS[867].EXT.AlarmWarnUnAck := FALSE;
   STATUS[867].EXT.AckRequired := FALSE;
   STATUS[867].EXT.Maintanence := FALSE;
   STATUS[867].EXT.Operation := FALSE;
   STATUS[867].EXT.Forced := FALSE;
   STATUS[867].EXT.BIT29 := FALSE;
   STATUS[867].EXT.BIT30 := FALSE;
   STATUS[867].EXT.BIT31 := FALSE;
   STATUS[867].EXT.ModeBit1 := FALSE;
   STATUS[867].EXT.ModeBit2 := FALSE;
   STATUS[867].EXT.ModeBit3 := FALSE;
   STATUS[867].EXT.BIT19 := FALSE;
   STATUS[867].EXT.BIT20 := FALSE;
   STATUS[867].EXT.AlarmSuppressed := FALSE;
   STATUS[867].EXT.AlarmPresent := FALSE;
   STATUS[867].EXT.AlarmFailUnAck := FALSE;
   STATUS[867].Status := 0;
   STATUS[867].TimeStamp := 16#0000;
   STATUS[868].EXT.AlarmWarnUnAck := FALSE;
   STATUS[868].EXT.AckRequired := FALSE;
   STATUS[868].EXT.Maintanence := FALSE;
   STATUS[868].EXT.Operation := FALSE;
   STATUS[868].EXT.Forced := FALSE;
   STATUS[868].EXT.BIT29 := FALSE;
   STATUS[868].EXT.BIT30 := FALSE;
   STATUS[868].EXT.BIT31 := FALSE;
   STATUS[868].EXT.ModeBit1 := FALSE;
   STATUS[868].EXT.ModeBit2 := FALSE;
   STATUS[868].EXT.ModeBit3 := FALSE;
   STATUS[868].EXT.BIT19 := FALSE;
   STATUS[868].EXT.BIT20 := FALSE;
   STATUS[868].EXT.AlarmSuppressed := FALSE;
   STATUS[868].EXT.AlarmPresent := FALSE;
   STATUS[868].EXT.AlarmFailUnAck := FALSE;
   STATUS[868].Status := 0;
   STATUS[868].TimeStamp := 16#0000;
   STATUS[869].EXT.AlarmWarnUnAck := FALSE;
   STATUS[869].EXT.AckRequired := FALSE;
   STATUS[869].EXT.Maintanence := FALSE;
   STATUS[869].EXT.Operation := FALSE;
   STATUS[869].EXT.Forced := FALSE;
   STATUS[869].EXT.BIT29 := FALSE;
   STATUS[869].EXT.BIT30 := FALSE;
   STATUS[869].EXT.BIT31 := FALSE;
   STATUS[869].EXT.ModeBit1 := FALSE;
   STATUS[869].EXT.ModeBit2 := FALSE;
   STATUS[869].EXT.ModeBit3 := FALSE;
   STATUS[869].EXT.BIT19 := FALSE;
   STATUS[869].EXT.BIT20 := FALSE;
   STATUS[869].EXT.AlarmSuppressed := FALSE;
   STATUS[869].EXT.AlarmPresent := FALSE;
   STATUS[869].EXT.AlarmFailUnAck := FALSE;
   STATUS[869].Status := 0;
   STATUS[869].TimeStamp := 16#0000;
   STATUS[870].EXT.AlarmWarnUnAck := FALSE;
   STATUS[870].EXT.AckRequired := FALSE;
   STATUS[870].EXT.Maintanence := FALSE;
   STATUS[870].EXT.Operation := FALSE;
   STATUS[870].EXT.Forced := FALSE;
   STATUS[870].EXT.BIT29 := FALSE;
   STATUS[870].EXT.BIT30 := FALSE;
   STATUS[870].EXT.BIT31 := FALSE;
   STATUS[870].EXT.ModeBit1 := FALSE;
   STATUS[870].EXT.ModeBit2 := FALSE;
   STATUS[870].EXT.ModeBit3 := FALSE;
   STATUS[870].EXT.BIT19 := FALSE;
   STATUS[870].EXT.BIT20 := FALSE;
   STATUS[870].EXT.AlarmSuppressed := FALSE;
   STATUS[870].EXT.AlarmPresent := FALSE;
   STATUS[870].EXT.AlarmFailUnAck := FALSE;
   STATUS[870].Status := 0;
   STATUS[870].TimeStamp := 16#0000;
   STATUS[871].EXT.AlarmWarnUnAck := FALSE;
   STATUS[871].EXT.AckRequired := FALSE;
   STATUS[871].EXT.Maintanence := FALSE;
   STATUS[871].EXT.Operation := FALSE;
   STATUS[871].EXT.Forced := FALSE;
   STATUS[871].EXT.BIT29 := FALSE;
   STATUS[871].EXT.BIT30 := FALSE;
   STATUS[871].EXT.BIT31 := FALSE;
   STATUS[871].EXT.ModeBit1 := FALSE;
   STATUS[871].EXT.ModeBit2 := FALSE;
   STATUS[871].EXT.ModeBit3 := FALSE;
   STATUS[871].EXT.BIT19 := FALSE;
   STATUS[871].EXT.BIT20 := FALSE;
   STATUS[871].EXT.AlarmSuppressed := FALSE;
   STATUS[871].EXT.AlarmPresent := FALSE;
   STATUS[871].EXT.AlarmFailUnAck := FALSE;
   STATUS[871].Status := 0;
   STATUS[871].TimeStamp := 16#0000;
   STATUS[872].EXT.AlarmWarnUnAck := FALSE;
   STATUS[872].EXT.AckRequired := FALSE;
   STATUS[872].EXT.Maintanence := FALSE;
   STATUS[872].EXT.Operation := FALSE;
   STATUS[872].EXT.Forced := FALSE;
   STATUS[872].EXT.BIT29 := FALSE;
   STATUS[872].EXT.BIT30 := FALSE;
   STATUS[872].EXT.BIT31 := FALSE;
   STATUS[872].EXT.ModeBit1 := FALSE;
   STATUS[872].EXT.ModeBit2 := FALSE;
   STATUS[872].EXT.ModeBit3 := FALSE;
   STATUS[872].EXT.BIT19 := FALSE;
   STATUS[872].EXT.BIT20 := FALSE;
   STATUS[872].EXT.AlarmSuppressed := FALSE;
   STATUS[872].EXT.AlarmPresent := FALSE;
   STATUS[872].EXT.AlarmFailUnAck := FALSE;
   STATUS[872].Status := 0;
   STATUS[872].TimeStamp := 16#0000;
   STATUS[873].EXT.AlarmWarnUnAck := FALSE;
   STATUS[873].EXT.AckRequired := FALSE;
   STATUS[873].EXT.Maintanence := FALSE;
   STATUS[873].EXT.Operation := FALSE;
   STATUS[873].EXT.Forced := FALSE;
   STATUS[873].EXT.BIT29 := FALSE;
   STATUS[873].EXT.BIT30 := FALSE;
   STATUS[873].EXT.BIT31 := FALSE;
   STATUS[873].EXT.ModeBit1 := FALSE;
   STATUS[873].EXT.ModeBit2 := FALSE;
   STATUS[873].EXT.ModeBit3 := FALSE;
   STATUS[873].EXT.BIT19 := FALSE;
   STATUS[873].EXT.BIT20 := FALSE;
   STATUS[873].EXT.AlarmSuppressed := FALSE;
   STATUS[873].EXT.AlarmPresent := FALSE;
   STATUS[873].EXT.AlarmFailUnAck := FALSE;
   STATUS[873].Status := 0;
   STATUS[873].TimeStamp := 16#0000;
   STATUS[874].EXT.AlarmWarnUnAck := FALSE;
   STATUS[874].EXT.AckRequired := FALSE;
   STATUS[874].EXT.Maintanence := FALSE;
   STATUS[874].EXT.Operation := FALSE;
   STATUS[874].EXT.Forced := FALSE;
   STATUS[874].EXT.BIT29 := FALSE;
   STATUS[874].EXT.BIT30 := FALSE;
   STATUS[874].EXT.BIT31 := FALSE;
   STATUS[874].EXT.ModeBit1 := FALSE;
   STATUS[874].EXT.ModeBit2 := FALSE;
   STATUS[874].EXT.ModeBit3 := FALSE;
   STATUS[874].EXT.BIT19 := FALSE;
   STATUS[874].EXT.BIT20 := FALSE;
   STATUS[874].EXT.AlarmSuppressed := FALSE;
   STATUS[874].EXT.AlarmPresent := FALSE;
   STATUS[874].EXT.AlarmFailUnAck := FALSE;
   STATUS[874].Status := 0;
   STATUS[874].TimeStamp := 16#0000;
   STATUS[875].EXT.AlarmWarnUnAck := FALSE;
   STATUS[875].EXT.AckRequired := FALSE;
   STATUS[875].EXT.Maintanence := FALSE;
   STATUS[875].EXT.Operation := FALSE;
   STATUS[875].EXT.Forced := FALSE;
   STATUS[875].EXT.BIT29 := FALSE;
   STATUS[875].EXT.BIT30 := FALSE;
   STATUS[875].EXT.BIT31 := FALSE;
   STATUS[875].EXT.ModeBit1 := FALSE;
   STATUS[875].EXT.ModeBit2 := FALSE;
   STATUS[875].EXT.ModeBit3 := FALSE;
   STATUS[875].EXT.BIT19 := FALSE;
   STATUS[875].EXT.BIT20 := FALSE;
   STATUS[875].EXT.AlarmSuppressed := FALSE;
   STATUS[875].EXT.AlarmPresent := FALSE;
   STATUS[875].EXT.AlarmFailUnAck := FALSE;
   STATUS[875].Status := 0;
   STATUS[875].TimeStamp := 16#0000;
   STATUS[876].EXT.AlarmWarnUnAck := FALSE;
   STATUS[876].EXT.AckRequired := FALSE;
   STATUS[876].EXT.Maintanence := FALSE;
   STATUS[876].EXT.Operation := FALSE;
   STATUS[876].EXT.Forced := FALSE;
   STATUS[876].EXT.BIT29 := FALSE;
   STATUS[876].EXT.BIT30 := FALSE;
   STATUS[876].EXT.BIT31 := FALSE;
   STATUS[876].EXT.ModeBit1 := FALSE;
   STATUS[876].EXT.ModeBit2 := FALSE;
   STATUS[876].EXT.ModeBit3 := FALSE;
   STATUS[876].EXT.BIT19 := FALSE;
   STATUS[876].EXT.BIT20 := FALSE;
   STATUS[876].EXT.AlarmSuppressed := FALSE;
   STATUS[876].EXT.AlarmPresent := FALSE;
   STATUS[876].EXT.AlarmFailUnAck := FALSE;
   STATUS[876].Status := 0;
   STATUS[876].TimeStamp := 16#0000;
   STATUS[877].EXT.AlarmWarnUnAck := FALSE;
   STATUS[877].EXT.AckRequired := FALSE;
   STATUS[877].EXT.Maintanence := FALSE;
   STATUS[877].EXT.Operation := FALSE;
   STATUS[877].EXT.Forced := FALSE;
   STATUS[877].EXT.BIT29 := FALSE;
   STATUS[877].EXT.BIT30 := FALSE;
   STATUS[877].EXT.BIT31 := FALSE;
   STATUS[877].EXT.ModeBit1 := FALSE;
   STATUS[877].EXT.ModeBit2 := FALSE;
   STATUS[877].EXT.ModeBit3 := FALSE;
   STATUS[877].EXT.BIT19 := FALSE;
   STATUS[877].EXT.BIT20 := FALSE;
   STATUS[877].EXT.AlarmSuppressed := FALSE;
   STATUS[877].EXT.AlarmPresent := FALSE;
   STATUS[877].EXT.AlarmFailUnAck := FALSE;
   STATUS[877].Status := 0;
   STATUS[877].TimeStamp := 16#0000;
   STATUS[878].EXT.AlarmWarnUnAck := FALSE;
   STATUS[878].EXT.AckRequired := FALSE;
   STATUS[878].EXT.Maintanence := FALSE;
   STATUS[878].EXT.Operation := FALSE;
   STATUS[878].EXT.Forced := FALSE;
   STATUS[878].EXT.BIT29 := FALSE;
   STATUS[878].EXT.BIT30 := FALSE;
   STATUS[878].EXT.BIT31 := FALSE;
   STATUS[878].EXT.ModeBit1 := FALSE;
   STATUS[878].EXT.ModeBit2 := FALSE;
   STATUS[878].EXT.ModeBit3 := FALSE;
   STATUS[878].EXT.BIT19 := FALSE;
   STATUS[878].EXT.BIT20 := FALSE;
   STATUS[878].EXT.AlarmSuppressed := FALSE;
   STATUS[878].EXT.AlarmPresent := FALSE;
   STATUS[878].EXT.AlarmFailUnAck := FALSE;
   STATUS[878].Status := 0;
   STATUS[878].TimeStamp := 16#0000;
   STATUS[879].EXT.AlarmWarnUnAck := FALSE;
   STATUS[879].EXT.AckRequired := FALSE;
   STATUS[879].EXT.Maintanence := FALSE;
   STATUS[879].EXT.Operation := FALSE;
   STATUS[879].EXT.Forced := FALSE;
   STATUS[879].EXT.BIT29 := FALSE;
   STATUS[879].EXT.BIT30 := FALSE;
   STATUS[879].EXT.BIT31 := FALSE;
   STATUS[879].EXT.ModeBit1 := FALSE;
   STATUS[879].EXT.ModeBit2 := FALSE;
   STATUS[879].EXT.ModeBit3 := FALSE;
   STATUS[879].EXT.BIT19 := FALSE;
   STATUS[879].EXT.BIT20 := FALSE;
   STATUS[879].EXT.AlarmSuppressed := FALSE;
   STATUS[879].EXT.AlarmPresent := FALSE;
   STATUS[879].EXT.AlarmFailUnAck := FALSE;
   STATUS[879].Status := 0;
   STATUS[879].TimeStamp := 16#0000;
   STATUS[880].EXT.AlarmWarnUnAck := FALSE;
   STATUS[880].EXT.AckRequired := FALSE;
   STATUS[880].EXT.Maintanence := FALSE;
   STATUS[880].EXT.Operation := FALSE;
   STATUS[880].EXT.Forced := FALSE;
   STATUS[880].EXT.BIT29 := FALSE;
   STATUS[880].EXT.BIT30 := FALSE;
   STATUS[880].EXT.BIT31 := FALSE;
   STATUS[880].EXT.ModeBit1 := FALSE;
   STATUS[880].EXT.ModeBit2 := FALSE;
   STATUS[880].EXT.ModeBit3 := FALSE;
   STATUS[880].EXT.BIT19 := FALSE;
   STATUS[880].EXT.BIT20 := FALSE;
   STATUS[880].EXT.AlarmSuppressed := FALSE;
   STATUS[880].EXT.AlarmPresent := FALSE;
   STATUS[880].EXT.AlarmFailUnAck := FALSE;
   STATUS[880].Status := 0;
   STATUS[880].TimeStamp := 16#0000;
   STATUS[881].EXT.AlarmWarnUnAck := FALSE;
   STATUS[881].EXT.AckRequired := FALSE;
   STATUS[881].EXT.Maintanence := FALSE;
   STATUS[881].EXT.Operation := FALSE;
   STATUS[881].EXT.Forced := FALSE;
   STATUS[881].EXT.BIT29 := FALSE;
   STATUS[881].EXT.BIT30 := FALSE;
   STATUS[881].EXT.BIT31 := FALSE;
   STATUS[881].EXT.ModeBit1 := FALSE;
   STATUS[881].EXT.ModeBit2 := FALSE;
   STATUS[881].EXT.ModeBit3 := FALSE;
   STATUS[881].EXT.BIT19 := FALSE;
   STATUS[881].EXT.BIT20 := FALSE;
   STATUS[881].EXT.AlarmSuppressed := FALSE;
   STATUS[881].EXT.AlarmPresent := FALSE;
   STATUS[881].EXT.AlarmFailUnAck := FALSE;
   STATUS[881].Status := 0;
   STATUS[881].TimeStamp := 16#0000;
   STATUS[882].EXT.AlarmWarnUnAck := FALSE;
   STATUS[882].EXT.AckRequired := FALSE;
   STATUS[882].EXT.Maintanence := FALSE;
   STATUS[882].EXT.Operation := FALSE;
   STATUS[882].EXT.Forced := FALSE;
   STATUS[882].EXT.BIT29 := FALSE;
   STATUS[882].EXT.BIT30 := FALSE;
   STATUS[882].EXT.BIT31 := FALSE;
   STATUS[882].EXT.ModeBit1 := FALSE;
   STATUS[882].EXT.ModeBit2 := FALSE;
   STATUS[882].EXT.ModeBit3 := FALSE;
   STATUS[882].EXT.BIT19 := FALSE;
   STATUS[882].EXT.BIT20 := FALSE;
   STATUS[882].EXT.AlarmSuppressed := FALSE;
   STATUS[882].EXT.AlarmPresent := FALSE;
   STATUS[882].EXT.AlarmFailUnAck := FALSE;
   STATUS[882].Status := 0;
   STATUS[882].TimeStamp := 16#0000;
   STATUS[883].EXT.AlarmWarnUnAck := FALSE;
   STATUS[883].EXT.AckRequired := FALSE;
   STATUS[883].EXT.Maintanence := FALSE;
   STATUS[883].EXT.Operation := FALSE;
   STATUS[883].EXT.Forced := FALSE;
   STATUS[883].EXT.BIT29 := FALSE;
   STATUS[883].EXT.BIT30 := FALSE;
   STATUS[883].EXT.BIT31 := FALSE;
   STATUS[883].EXT.ModeBit1 := FALSE;
   STATUS[883].EXT.ModeBit2 := FALSE;
   STATUS[883].EXT.ModeBit3 := FALSE;
   STATUS[883].EXT.BIT19 := FALSE;
   STATUS[883].EXT.BIT20 := FALSE;
   STATUS[883].EXT.AlarmSuppressed := FALSE;
   STATUS[883].EXT.AlarmPresent := FALSE;
   STATUS[883].EXT.AlarmFailUnAck := FALSE;
   STATUS[883].Status := 0;
   STATUS[883].TimeStamp := 16#0000;
   STATUS[884].EXT.AlarmWarnUnAck := FALSE;
   STATUS[884].EXT.AckRequired := FALSE;
   STATUS[884].EXT.Maintanence := FALSE;
   STATUS[884].EXT.Operation := FALSE;
   STATUS[884].EXT.Forced := FALSE;
   STATUS[884].EXT.BIT29 := FALSE;
   STATUS[884].EXT.BIT30 := FALSE;
   STATUS[884].EXT.BIT31 := FALSE;
   STATUS[884].EXT.ModeBit1 := FALSE;
   STATUS[884].EXT.ModeBit2 := FALSE;
   STATUS[884].EXT.ModeBit3 := FALSE;
   STATUS[884].EXT.BIT19 := FALSE;
   STATUS[884].EXT.BIT20 := FALSE;
   STATUS[884].EXT.AlarmSuppressed := FALSE;
   STATUS[884].EXT.AlarmPresent := FALSE;
   STATUS[884].EXT.AlarmFailUnAck := FALSE;
   STATUS[884].Status := 0;
   STATUS[884].TimeStamp := 16#0000;
   STATUS[885].EXT.AlarmWarnUnAck := FALSE;
   STATUS[885].EXT.AckRequired := FALSE;
   STATUS[885].EXT.Maintanence := FALSE;
   STATUS[885].EXT.Operation := FALSE;
   STATUS[885].EXT.Forced := FALSE;
   STATUS[885].EXT.BIT29 := FALSE;
   STATUS[885].EXT.BIT30 := FALSE;
   STATUS[885].EXT.BIT31 := FALSE;
   STATUS[885].EXT.ModeBit1 := FALSE;
   STATUS[885].EXT.ModeBit2 := FALSE;
   STATUS[885].EXT.ModeBit3 := FALSE;
   STATUS[885].EXT.BIT19 := FALSE;
   STATUS[885].EXT.BIT20 := FALSE;
   STATUS[885].EXT.AlarmSuppressed := FALSE;
   STATUS[885].EXT.AlarmPresent := FALSE;
   STATUS[885].EXT.AlarmFailUnAck := FALSE;
   STATUS[885].Status := 0;
   STATUS[885].TimeStamp := 16#0000;
   STATUS[886].EXT.AlarmWarnUnAck := FALSE;
   STATUS[886].EXT.AckRequired := FALSE;
   STATUS[886].EXT.Maintanence := FALSE;
   STATUS[886].EXT.Operation := FALSE;
   STATUS[886].EXT.Forced := FALSE;
   STATUS[886].EXT.BIT29 := FALSE;
   STATUS[886].EXT.BIT30 := FALSE;
   STATUS[886].EXT.BIT31 := FALSE;
   STATUS[886].EXT.ModeBit1 := FALSE;
   STATUS[886].EXT.ModeBit2 := FALSE;
   STATUS[886].EXT.ModeBit3 := FALSE;
   STATUS[886].EXT.BIT19 := FALSE;
   STATUS[886].EXT.BIT20 := FALSE;
   STATUS[886].EXT.AlarmSuppressed := FALSE;
   STATUS[886].EXT.AlarmPresent := FALSE;
   STATUS[886].EXT.AlarmFailUnAck := FALSE;
   STATUS[886].Status := 0;
   STATUS[886].TimeStamp := 16#0000;
   STATUS[887].EXT.AlarmWarnUnAck := FALSE;
   STATUS[887].EXT.AckRequired := FALSE;
   STATUS[887].EXT.Maintanence := FALSE;
   STATUS[887].EXT.Operation := FALSE;
   STATUS[887].EXT.Forced := FALSE;
   STATUS[887].EXT.BIT29 := FALSE;
   STATUS[887].EXT.BIT30 := FALSE;
   STATUS[887].EXT.BIT31 := FALSE;
   STATUS[887].EXT.ModeBit1 := FALSE;
   STATUS[887].EXT.ModeBit2 := FALSE;
   STATUS[887].EXT.ModeBit3 := FALSE;
   STATUS[887].EXT.BIT19 := FALSE;
   STATUS[887].EXT.BIT20 := FALSE;
   STATUS[887].EXT.AlarmSuppressed := FALSE;
   STATUS[887].EXT.AlarmPresent := FALSE;
   STATUS[887].EXT.AlarmFailUnAck := FALSE;
   STATUS[887].Status := 0;
   STATUS[887].TimeStamp := 16#0000;
   STATUS[888].EXT.AlarmWarnUnAck := FALSE;
   STATUS[888].EXT.AckRequired := FALSE;
   STATUS[888].EXT.Maintanence := FALSE;
   STATUS[888].EXT.Operation := FALSE;
   STATUS[888].EXT.Forced := FALSE;
   STATUS[888].EXT.BIT29 := FALSE;
   STATUS[888].EXT.BIT30 := FALSE;
   STATUS[888].EXT.BIT31 := FALSE;
   STATUS[888].EXT.ModeBit1 := FALSE;
   STATUS[888].EXT.ModeBit2 := FALSE;
   STATUS[888].EXT.ModeBit3 := FALSE;
   STATUS[888].EXT.BIT19 := FALSE;
   STATUS[888].EXT.BIT20 := FALSE;
   STATUS[888].EXT.AlarmSuppressed := FALSE;
   STATUS[888].EXT.AlarmPresent := FALSE;
   STATUS[888].EXT.AlarmFailUnAck := FALSE;
   STATUS[888].Status := 0;
   STATUS[888].TimeStamp := 16#0000;
   STATUS[889].EXT.AlarmWarnUnAck := FALSE;
   STATUS[889].EXT.AckRequired := FALSE;
   STATUS[889].EXT.Maintanence := FALSE;
   STATUS[889].EXT.Operation := FALSE;
   STATUS[889].EXT.Forced := FALSE;
   STATUS[889].EXT.BIT29 := FALSE;
   STATUS[889].EXT.BIT30 := FALSE;
   STATUS[889].EXT.BIT31 := FALSE;
   STATUS[889].EXT.ModeBit1 := FALSE;
   STATUS[889].EXT.ModeBit2 := FALSE;
   STATUS[889].EXT.ModeBit3 := FALSE;
   STATUS[889].EXT.BIT19 := FALSE;
   STATUS[889].EXT.BIT20 := FALSE;
   STATUS[889].EXT.AlarmSuppressed := FALSE;
   STATUS[889].EXT.AlarmPresent := FALSE;
   STATUS[889].EXT.AlarmFailUnAck := FALSE;
   STATUS[889].Status := 0;
   STATUS[889].TimeStamp := 16#0000;
   STATUS[890].EXT.AlarmWarnUnAck := FALSE;
   STATUS[890].EXT.AckRequired := FALSE;
   STATUS[890].EXT.Maintanence := FALSE;
   STATUS[890].EXT.Operation := FALSE;
   STATUS[890].EXT.Forced := FALSE;
   STATUS[890].EXT.BIT29 := FALSE;
   STATUS[890].EXT.BIT30 := FALSE;
   STATUS[890].EXT.BIT31 := FALSE;
   STATUS[890].EXT.ModeBit1 := FALSE;
   STATUS[890].EXT.ModeBit2 := FALSE;
   STATUS[890].EXT.ModeBit3 := FALSE;
   STATUS[890].EXT.BIT19 := FALSE;
   STATUS[890].EXT.BIT20 := FALSE;
   STATUS[890].EXT.AlarmSuppressed := FALSE;
   STATUS[890].EXT.AlarmPresent := FALSE;
   STATUS[890].EXT.AlarmFailUnAck := FALSE;
   STATUS[890].Status := 0;
   STATUS[890].TimeStamp := 16#0000;
   STATUS[891].EXT.AlarmWarnUnAck := FALSE;
   STATUS[891].EXT.AckRequired := FALSE;
   STATUS[891].EXT.Maintanence := FALSE;
   STATUS[891].EXT.Operation := FALSE;
   STATUS[891].EXT.Forced := FALSE;
   STATUS[891].EXT.BIT29 := FALSE;
   STATUS[891].EXT.BIT30 := FALSE;
   STATUS[891].EXT.BIT31 := FALSE;
   STATUS[891].EXT.ModeBit1 := FALSE;
   STATUS[891].EXT.ModeBit2 := FALSE;
   STATUS[891].EXT.ModeBit3 := FALSE;
   STATUS[891].EXT.BIT19 := FALSE;
   STATUS[891].EXT.BIT20 := FALSE;
   STATUS[891].EXT.AlarmSuppressed := FALSE;
   STATUS[891].EXT.AlarmPresent := FALSE;
   STATUS[891].EXT.AlarmFailUnAck := FALSE;
   STATUS[891].Status := 0;
   STATUS[891].TimeStamp := 16#0000;
   STATUS[892].EXT.AlarmWarnUnAck := FALSE;
   STATUS[892].EXT.AckRequired := FALSE;
   STATUS[892].EXT.Maintanence := FALSE;
   STATUS[892].EXT.Operation := FALSE;
   STATUS[892].EXT.Forced := FALSE;
   STATUS[892].EXT.BIT29 := FALSE;
   STATUS[892].EXT.BIT30 := FALSE;
   STATUS[892].EXT.BIT31 := FALSE;
   STATUS[892].EXT.ModeBit1 := FALSE;
   STATUS[892].EXT.ModeBit2 := FALSE;
   STATUS[892].EXT.ModeBit3 := FALSE;
   STATUS[892].EXT.BIT19 := FALSE;
   STATUS[892].EXT.BIT20 := FALSE;
   STATUS[892].EXT.AlarmSuppressed := FALSE;
   STATUS[892].EXT.AlarmPresent := FALSE;
   STATUS[892].EXT.AlarmFailUnAck := FALSE;
   STATUS[892].Status := 0;
   STATUS[892].TimeStamp := 16#0000;
   STATUS[893].EXT.AlarmWarnUnAck := FALSE;
   STATUS[893].EXT.AckRequired := FALSE;
   STATUS[893].EXT.Maintanence := FALSE;
   STATUS[893].EXT.Operation := FALSE;
   STATUS[893].EXT.Forced := FALSE;
   STATUS[893].EXT.BIT29 := FALSE;
   STATUS[893].EXT.BIT30 := FALSE;
   STATUS[893].EXT.BIT31 := FALSE;
   STATUS[893].EXT.ModeBit1 := FALSE;
   STATUS[893].EXT.ModeBit2 := FALSE;
   STATUS[893].EXT.ModeBit3 := FALSE;
   STATUS[893].EXT.BIT19 := FALSE;
   STATUS[893].EXT.BIT20 := FALSE;
   STATUS[893].EXT.AlarmSuppressed := FALSE;
   STATUS[893].EXT.AlarmPresent := FALSE;
   STATUS[893].EXT.AlarmFailUnAck := FALSE;
   STATUS[893].Status := 0;
   STATUS[893].TimeStamp := 16#0000;
   STATUS[894].EXT.AlarmWarnUnAck := FALSE;
   STATUS[894].EXT.AckRequired := FALSE;
   STATUS[894].EXT.Maintanence := FALSE;
   STATUS[894].EXT.Operation := FALSE;
   STATUS[894].EXT.Forced := FALSE;
   STATUS[894].EXT.BIT29 := FALSE;
   STATUS[894].EXT.BIT30 := FALSE;
   STATUS[894].EXT.BIT31 := FALSE;
   STATUS[894].EXT.ModeBit1 := FALSE;
   STATUS[894].EXT.ModeBit2 := FALSE;
   STATUS[894].EXT.ModeBit3 := FALSE;
   STATUS[894].EXT.BIT19 := FALSE;
   STATUS[894].EXT.BIT20 := FALSE;
   STATUS[894].EXT.AlarmSuppressed := FALSE;
   STATUS[894].EXT.AlarmPresent := FALSE;
   STATUS[894].EXT.AlarmFailUnAck := FALSE;
   STATUS[894].Status := 0;
   STATUS[894].TimeStamp := 16#0000;
   STATUS[895].EXT.AlarmWarnUnAck := FALSE;
   STATUS[895].EXT.AckRequired := FALSE;
   STATUS[895].EXT.Maintanence := FALSE;
   STATUS[895].EXT.Operation := FALSE;
   STATUS[895].EXT.Forced := FALSE;
   STATUS[895].EXT.BIT29 := FALSE;
   STATUS[895].EXT.BIT30 := FALSE;
   STATUS[895].EXT.BIT31 := FALSE;
   STATUS[895].EXT.ModeBit1 := FALSE;
   STATUS[895].EXT.ModeBit2 := FALSE;
   STATUS[895].EXT.ModeBit3 := FALSE;
   STATUS[895].EXT.BIT19 := FALSE;
   STATUS[895].EXT.BIT20 := FALSE;
   STATUS[895].EXT.AlarmSuppressed := FALSE;
   STATUS[895].EXT.AlarmPresent := FALSE;
   STATUS[895].EXT.AlarmFailUnAck := FALSE;
   STATUS[895].Status := 0;
   STATUS[895].TimeStamp := 16#0000;
   STATUS[896].EXT.AlarmWarnUnAck := FALSE;
   STATUS[896].EXT.AckRequired := FALSE;
   STATUS[896].EXT.Maintanence := FALSE;
   STATUS[896].EXT.Operation := FALSE;
   STATUS[896].EXT.Forced := FALSE;
   STATUS[896].EXT.BIT29 := FALSE;
   STATUS[896].EXT.BIT30 := FALSE;
   STATUS[896].EXT.BIT31 := FALSE;
   STATUS[896].EXT.ModeBit1 := FALSE;
   STATUS[896].EXT.ModeBit2 := FALSE;
   STATUS[896].EXT.ModeBit3 := FALSE;
   STATUS[896].EXT.BIT19 := FALSE;
   STATUS[896].EXT.BIT20 := FALSE;
   STATUS[896].EXT.AlarmSuppressed := FALSE;
   STATUS[896].EXT.AlarmPresent := FALSE;
   STATUS[896].EXT.AlarmFailUnAck := FALSE;
   STATUS[896].Status := 0;
   STATUS[896].TimeStamp := 16#0000;
   STATUS[897].EXT.AlarmWarnUnAck := FALSE;
   STATUS[897].EXT.AckRequired := FALSE;
   STATUS[897].EXT.Maintanence := FALSE;
   STATUS[897].EXT.Operation := FALSE;
   STATUS[897].EXT.Forced := FALSE;
   STATUS[897].EXT.BIT29 := FALSE;
   STATUS[897].EXT.BIT30 := FALSE;
   STATUS[897].EXT.BIT31 := FALSE;
   STATUS[897].EXT.ModeBit1 := FALSE;
   STATUS[897].EXT.ModeBit2 := FALSE;
   STATUS[897].EXT.ModeBit3 := FALSE;
   STATUS[897].EXT.BIT19 := FALSE;
   STATUS[897].EXT.BIT20 := FALSE;
   STATUS[897].EXT.AlarmSuppressed := FALSE;
   STATUS[897].EXT.AlarmPresent := FALSE;
   STATUS[897].EXT.AlarmFailUnAck := FALSE;
   STATUS[897].Status := 0;
   STATUS[897].TimeStamp := 16#0000;
   STATUS[898].EXT.AlarmWarnUnAck := FALSE;
   STATUS[898].EXT.AckRequired := FALSE;
   STATUS[898].EXT.Maintanence := FALSE;
   STATUS[898].EXT.Operation := FALSE;
   STATUS[898].EXT.Forced := FALSE;
   STATUS[898].EXT.BIT29 := FALSE;
   STATUS[898].EXT.BIT30 := FALSE;
   STATUS[898].EXT.BIT31 := FALSE;
   STATUS[898].EXT.ModeBit1 := FALSE;
   STATUS[898].EXT.ModeBit2 := FALSE;
   STATUS[898].EXT.ModeBit3 := FALSE;
   STATUS[898].EXT.BIT19 := FALSE;
   STATUS[898].EXT.BIT20 := FALSE;
   STATUS[898].EXT.AlarmSuppressed := FALSE;
   STATUS[898].EXT.AlarmPresent := FALSE;
   STATUS[898].EXT.AlarmFailUnAck := FALSE;
   STATUS[898].Status := 0;
   STATUS[898].TimeStamp := 16#0000;
   STATUS[899].EXT.AlarmWarnUnAck := FALSE;
   STATUS[899].EXT.AckRequired := FALSE;
   STATUS[899].EXT.Maintanence := FALSE;
   STATUS[899].EXT.Operation := FALSE;
   STATUS[899].EXT.Forced := FALSE;
   STATUS[899].EXT.BIT29 := FALSE;
   STATUS[899].EXT.BIT30 := FALSE;
   STATUS[899].EXT.BIT31 := FALSE;
   STATUS[899].EXT.ModeBit1 := FALSE;
   STATUS[899].EXT.ModeBit2 := FALSE;
   STATUS[899].EXT.ModeBit3 := FALSE;
   STATUS[899].EXT.BIT19 := FALSE;
   STATUS[899].EXT.BIT20 := FALSE;
   STATUS[899].EXT.AlarmSuppressed := FALSE;
   STATUS[899].EXT.AlarmPresent := FALSE;
   STATUS[899].EXT.AlarmFailUnAck := FALSE;
   STATUS[899].Status := 0;
   STATUS[899].TimeStamp := 16#0000;
   STATUS[900].EXT.AlarmWarnUnAck := FALSE;
   STATUS[900].EXT.AckRequired := FALSE;
   STATUS[900].EXT.Maintanence := FALSE;
   STATUS[900].EXT.Operation := FALSE;
   STATUS[900].EXT.Forced := FALSE;
   STATUS[900].EXT.BIT29 := FALSE;
   STATUS[900].EXT.BIT30 := FALSE;
   STATUS[900].EXT.BIT31 := FALSE;
   STATUS[900].EXT.ModeBit1 := FALSE;
   STATUS[900].EXT.ModeBit2 := FALSE;
   STATUS[900].EXT.ModeBit3 := FALSE;
   STATUS[900].EXT.BIT19 := FALSE;
   STATUS[900].EXT.BIT20 := FALSE;
   STATUS[900].EXT.AlarmSuppressed := FALSE;
   STATUS[900].EXT.AlarmPresent := FALSE;
   STATUS[900].EXT.AlarmFailUnAck := FALSE;
   STATUS[900].Status := 0;
   STATUS[900].TimeStamp := 16#0000;
   STATUS[901].EXT.AlarmWarnUnAck := FALSE;
   STATUS[901].EXT.AckRequired := FALSE;
   STATUS[901].EXT.Maintanence := FALSE;
   STATUS[901].EXT.Operation := FALSE;
   STATUS[901].EXT.Forced := FALSE;
   STATUS[901].EXT.BIT29 := FALSE;
   STATUS[901].EXT.BIT30 := FALSE;
   STATUS[901].EXT.BIT31 := FALSE;
   STATUS[901].EXT.ModeBit1 := FALSE;
   STATUS[901].EXT.ModeBit2 := FALSE;
   STATUS[901].EXT.ModeBit3 := FALSE;
   STATUS[901].EXT.BIT19 := FALSE;
   STATUS[901].EXT.BIT20 := FALSE;
   STATUS[901].EXT.AlarmSuppressed := FALSE;
   STATUS[901].EXT.AlarmPresent := FALSE;
   STATUS[901].EXT.AlarmFailUnAck := FALSE;
   STATUS[901].Status := 0;
   STATUS[901].TimeStamp := 16#0000;
   STATUS[902].EXT.AlarmWarnUnAck := FALSE;
   STATUS[902].EXT.AckRequired := FALSE;
   STATUS[902].EXT.Maintanence := FALSE;
   STATUS[902].EXT.Operation := FALSE;
   STATUS[902].EXT.Forced := FALSE;
   STATUS[902].EXT.BIT29 := FALSE;
   STATUS[902].EXT.BIT30 := FALSE;
   STATUS[902].EXT.BIT31 := FALSE;
   STATUS[902].EXT.ModeBit1 := FALSE;
   STATUS[902].EXT.ModeBit2 := FALSE;
   STATUS[902].EXT.ModeBit3 := FALSE;
   STATUS[902].EXT.BIT19 := FALSE;
   STATUS[902].EXT.BIT20 := FALSE;
   STATUS[902].EXT.AlarmSuppressed := FALSE;
   STATUS[902].EXT.AlarmPresent := FALSE;
   STATUS[902].EXT.AlarmFailUnAck := FALSE;
   STATUS[902].Status := 0;
   STATUS[902].TimeStamp := 16#0000;
   STATUS[903].EXT.AlarmWarnUnAck := FALSE;
   STATUS[903].EXT.AckRequired := FALSE;
   STATUS[903].EXT.Maintanence := FALSE;
   STATUS[903].EXT.Operation := FALSE;
   STATUS[903].EXT.Forced := FALSE;
   STATUS[903].EXT.BIT29 := FALSE;
   STATUS[903].EXT.BIT30 := FALSE;
   STATUS[903].EXT.BIT31 := FALSE;
   STATUS[903].EXT.ModeBit1 := FALSE;
   STATUS[903].EXT.ModeBit2 := FALSE;
   STATUS[903].EXT.ModeBit3 := FALSE;
   STATUS[903].EXT.BIT19 := FALSE;
   STATUS[903].EXT.BIT20 := FALSE;
   STATUS[903].EXT.AlarmSuppressed := FALSE;
   STATUS[903].EXT.AlarmPresent := FALSE;
   STATUS[903].EXT.AlarmFailUnAck := FALSE;
   STATUS[903].Status := 0;
   STATUS[903].TimeStamp := 16#0000;
   STATUS[904].EXT.AlarmWarnUnAck := FALSE;
   STATUS[904].EXT.AckRequired := FALSE;
   STATUS[904].EXT.Maintanence := FALSE;
   STATUS[904].EXT.Operation := FALSE;
   STATUS[904].EXT.Forced := FALSE;
   STATUS[904].EXT.BIT29 := FALSE;
   STATUS[904].EXT.BIT30 := FALSE;
   STATUS[904].EXT.BIT31 := FALSE;
   STATUS[904].EXT.ModeBit1 := FALSE;
   STATUS[904].EXT.ModeBit2 := FALSE;
   STATUS[904].EXT.ModeBit3 := FALSE;
   STATUS[904].EXT.BIT19 := FALSE;
   STATUS[904].EXT.BIT20 := FALSE;
   STATUS[904].EXT.AlarmSuppressed := FALSE;
   STATUS[904].EXT.AlarmPresent := FALSE;
   STATUS[904].EXT.AlarmFailUnAck := FALSE;
   STATUS[904].Status := 0;
   STATUS[904].TimeStamp := 16#0000;
   STATUS[905].EXT.AlarmWarnUnAck := FALSE;
   STATUS[905].EXT.AckRequired := FALSE;
   STATUS[905].EXT.Maintanence := FALSE;
   STATUS[905].EXT.Operation := FALSE;
   STATUS[905].EXT.Forced := FALSE;
   STATUS[905].EXT.BIT29 := FALSE;
   STATUS[905].EXT.BIT30 := FALSE;
   STATUS[905].EXT.BIT31 := FALSE;
   STATUS[905].EXT.ModeBit1 := FALSE;
   STATUS[905].EXT.ModeBit2 := FALSE;
   STATUS[905].EXT.ModeBit3 := FALSE;
   STATUS[905].EXT.BIT19 := FALSE;
   STATUS[905].EXT.BIT20 := FALSE;
   STATUS[905].EXT.AlarmSuppressed := FALSE;
   STATUS[905].EXT.AlarmPresent := FALSE;
   STATUS[905].EXT.AlarmFailUnAck := FALSE;
   STATUS[905].Status := 0;
   STATUS[905].TimeStamp := 16#0000;
   STATUS[906].EXT.AlarmWarnUnAck := FALSE;
   STATUS[906].EXT.AckRequired := FALSE;
   STATUS[906].EXT.Maintanence := FALSE;
   STATUS[906].EXT.Operation := FALSE;
   STATUS[906].EXT.Forced := FALSE;
   STATUS[906].EXT.BIT29 := FALSE;
   STATUS[906].EXT.BIT30 := FALSE;
   STATUS[906].EXT.BIT31 := FALSE;
   STATUS[906].EXT.ModeBit1 := FALSE;
   STATUS[906].EXT.ModeBit2 := FALSE;
   STATUS[906].EXT.ModeBit3 := FALSE;
   STATUS[906].EXT.BIT19 := FALSE;
   STATUS[906].EXT.BIT20 := FALSE;
   STATUS[906].EXT.AlarmSuppressed := FALSE;
   STATUS[906].EXT.AlarmPresent := FALSE;
   STATUS[906].EXT.AlarmFailUnAck := FALSE;
   STATUS[906].Status := 0;
   STATUS[906].TimeStamp := 16#0000;
   STATUS[907].EXT.AlarmWarnUnAck := FALSE;
   STATUS[907].EXT.AckRequired := FALSE;
   STATUS[907].EXT.Maintanence := FALSE;
   STATUS[907].EXT.Operation := FALSE;
   STATUS[907].EXT.Forced := FALSE;
   STATUS[907].EXT.BIT29 := FALSE;
   STATUS[907].EXT.BIT30 := FALSE;
   STATUS[907].EXT.BIT31 := FALSE;
   STATUS[907].EXT.ModeBit1 := FALSE;
   STATUS[907].EXT.ModeBit2 := FALSE;
   STATUS[907].EXT.ModeBit3 := FALSE;
   STATUS[907].EXT.BIT19 := FALSE;
   STATUS[907].EXT.BIT20 := FALSE;
   STATUS[907].EXT.AlarmSuppressed := FALSE;
   STATUS[907].EXT.AlarmPresent := FALSE;
   STATUS[907].EXT.AlarmFailUnAck := FALSE;
   STATUS[907].Status := 0;
   STATUS[907].TimeStamp := 16#0000;
   STATUS[908].EXT.AlarmWarnUnAck := FALSE;
   STATUS[908].EXT.AckRequired := FALSE;
   STATUS[908].EXT.Maintanence := FALSE;
   STATUS[908].EXT.Operation := FALSE;
   STATUS[908].EXT.Forced := FALSE;
   STATUS[908].EXT.BIT29 := FALSE;
   STATUS[908].EXT.BIT30 := FALSE;
   STATUS[908].EXT.BIT31 := FALSE;
   STATUS[908].EXT.ModeBit1 := FALSE;
   STATUS[908].EXT.ModeBit2 := FALSE;
   STATUS[908].EXT.ModeBit3 := FALSE;
   STATUS[908].EXT.BIT19 := FALSE;
   STATUS[908].EXT.BIT20 := FALSE;
   STATUS[908].EXT.AlarmSuppressed := FALSE;
   STATUS[908].EXT.AlarmPresent := FALSE;
   STATUS[908].EXT.AlarmFailUnAck := FALSE;
   STATUS[908].Status := 0;
   STATUS[908].TimeStamp := 16#0000;
   STATUS[909].EXT.AlarmWarnUnAck := FALSE;
   STATUS[909].EXT.AckRequired := FALSE;
   STATUS[909].EXT.Maintanence := FALSE;
   STATUS[909].EXT.Operation := FALSE;
   STATUS[909].EXT.Forced := FALSE;
   STATUS[909].EXT.BIT29 := FALSE;
   STATUS[909].EXT.BIT30 := FALSE;
   STATUS[909].EXT.BIT31 := FALSE;
   STATUS[909].EXT.ModeBit1 := FALSE;
   STATUS[909].EXT.ModeBit2 := FALSE;
   STATUS[909].EXT.ModeBit3 := FALSE;
   STATUS[909].EXT.BIT19 := FALSE;
   STATUS[909].EXT.BIT20 := FALSE;
   STATUS[909].EXT.AlarmSuppressed := FALSE;
   STATUS[909].EXT.AlarmPresent := FALSE;
   STATUS[909].EXT.AlarmFailUnAck := FALSE;
   STATUS[909].Status := 0;
   STATUS[909].TimeStamp := 16#0000;
   STATUS[910].EXT.AlarmWarnUnAck := FALSE;
   STATUS[910].EXT.AckRequired := FALSE;
   STATUS[910].EXT.Maintanence := FALSE;
   STATUS[910].EXT.Operation := FALSE;
   STATUS[910].EXT.Forced := FALSE;
   STATUS[910].EXT.BIT29 := FALSE;
   STATUS[910].EXT.BIT30 := FALSE;
   STATUS[910].EXT.BIT31 := FALSE;
   STATUS[910].EXT.ModeBit1 := FALSE;
   STATUS[910].EXT.ModeBit2 := FALSE;
   STATUS[910].EXT.ModeBit3 := FALSE;
   STATUS[910].EXT.BIT19 := FALSE;
   STATUS[910].EXT.BIT20 := FALSE;
   STATUS[910].EXT.AlarmSuppressed := FALSE;
   STATUS[910].EXT.AlarmPresent := FALSE;
   STATUS[910].EXT.AlarmFailUnAck := FALSE;
   STATUS[910].Status := 0;
   STATUS[910].TimeStamp := 16#0000;
   STATUS[911].EXT.AlarmWarnUnAck := FALSE;
   STATUS[911].EXT.AckRequired := FALSE;
   STATUS[911].EXT.Maintanence := FALSE;
   STATUS[911].EXT.Operation := FALSE;
   STATUS[911].EXT.Forced := FALSE;
   STATUS[911].EXT.BIT29 := FALSE;
   STATUS[911].EXT.BIT30 := FALSE;
   STATUS[911].EXT.BIT31 := FALSE;
   STATUS[911].EXT.ModeBit1 := FALSE;
   STATUS[911].EXT.ModeBit2 := FALSE;
   STATUS[911].EXT.ModeBit3 := FALSE;
   STATUS[911].EXT.BIT19 := FALSE;
   STATUS[911].EXT.BIT20 := FALSE;
   STATUS[911].EXT.AlarmSuppressed := FALSE;
   STATUS[911].EXT.AlarmPresent := FALSE;
   STATUS[911].EXT.AlarmFailUnAck := FALSE;
   STATUS[911].Status := 0;
   STATUS[911].TimeStamp := 16#0000;
   STATUS[912].EXT.AlarmWarnUnAck := FALSE;
   STATUS[912].EXT.AckRequired := FALSE;
   STATUS[912].EXT.Maintanence := FALSE;
   STATUS[912].EXT.Operation := FALSE;
   STATUS[912].EXT.Forced := FALSE;
   STATUS[912].EXT.BIT29 := FALSE;
   STATUS[912].EXT.BIT30 := FALSE;
   STATUS[912].EXT.BIT31 := FALSE;
   STATUS[912].EXT.ModeBit1 := FALSE;
   STATUS[912].EXT.ModeBit2 := FALSE;
   STATUS[912].EXT.ModeBit3 := FALSE;
   STATUS[912].EXT.BIT19 := FALSE;
   STATUS[912].EXT.BIT20 := FALSE;
   STATUS[912].EXT.AlarmSuppressed := FALSE;
   STATUS[912].EXT.AlarmPresent := FALSE;
   STATUS[912].EXT.AlarmFailUnAck := FALSE;
   STATUS[912].Status := 0;
   STATUS[912].TimeStamp := 16#0000;
   STATUS[913].EXT.AlarmWarnUnAck := FALSE;
   STATUS[913].EXT.AckRequired := FALSE;
   STATUS[913].EXT.Maintanence := FALSE;
   STATUS[913].EXT.Operation := FALSE;
   STATUS[913].EXT.Forced := FALSE;
   STATUS[913].EXT.BIT29 := FALSE;
   STATUS[913].EXT.BIT30 := FALSE;
   STATUS[913].EXT.BIT31 := FALSE;
   STATUS[913].EXT.ModeBit1 := FALSE;
   STATUS[913].EXT.ModeBit2 := FALSE;
   STATUS[913].EXT.ModeBit3 := FALSE;
   STATUS[913].EXT.BIT19 := FALSE;
   STATUS[913].EXT.BIT20 := FALSE;
   STATUS[913].EXT.AlarmSuppressed := FALSE;
   STATUS[913].EXT.AlarmPresent := FALSE;
   STATUS[913].EXT.AlarmFailUnAck := FALSE;
   STATUS[913].Status := 0;
   STATUS[913].TimeStamp := 16#0000;
   STATUS[914].EXT.AlarmWarnUnAck := FALSE;
   STATUS[914].EXT.AckRequired := FALSE;
   STATUS[914].EXT.Maintanence := FALSE;
   STATUS[914].EXT.Operation := FALSE;
   STATUS[914].EXT.Forced := FALSE;
   STATUS[914].EXT.BIT29 := FALSE;
   STATUS[914].EXT.BIT30 := FALSE;
   STATUS[914].EXT.BIT31 := FALSE;
   STATUS[914].EXT.ModeBit1 := FALSE;
   STATUS[914].EXT.ModeBit2 := FALSE;
   STATUS[914].EXT.ModeBit3 := FALSE;
   STATUS[914].EXT.BIT19 := FALSE;
   STATUS[914].EXT.BIT20 := FALSE;
   STATUS[914].EXT.AlarmSuppressed := FALSE;
   STATUS[914].EXT.AlarmPresent := FALSE;
   STATUS[914].EXT.AlarmFailUnAck := FALSE;
   STATUS[914].Status := 0;
   STATUS[914].TimeStamp := 16#0000;
   STATUS[915].EXT.AlarmWarnUnAck := FALSE;
   STATUS[915].EXT.AckRequired := FALSE;
   STATUS[915].EXT.Maintanence := FALSE;
   STATUS[915].EXT.Operation := FALSE;
   STATUS[915].EXT.Forced := FALSE;
   STATUS[915].EXT.BIT29 := FALSE;
   STATUS[915].EXT.BIT30 := FALSE;
   STATUS[915].EXT.BIT31 := FALSE;
   STATUS[915].EXT.ModeBit1 := FALSE;
   STATUS[915].EXT.ModeBit2 := FALSE;
   STATUS[915].EXT.ModeBit3 := FALSE;
   STATUS[915].EXT.BIT19 := FALSE;
   STATUS[915].EXT.BIT20 := FALSE;
   STATUS[915].EXT.AlarmSuppressed := FALSE;
   STATUS[915].EXT.AlarmPresent := FALSE;
   STATUS[915].EXT.AlarmFailUnAck := FALSE;
   STATUS[915].Status := 0;
   STATUS[915].TimeStamp := 16#0000;
   STATUS[916].EXT.AlarmWarnUnAck := FALSE;
   STATUS[916].EXT.AckRequired := FALSE;
   STATUS[916].EXT.Maintanence := FALSE;
   STATUS[916].EXT.Operation := FALSE;
   STATUS[916].EXT.Forced := FALSE;
   STATUS[916].EXT.BIT29 := FALSE;
   STATUS[916].EXT.BIT30 := FALSE;
   STATUS[916].EXT.BIT31 := FALSE;
   STATUS[916].EXT.ModeBit1 := FALSE;
   STATUS[916].EXT.ModeBit2 := FALSE;
   STATUS[916].EXT.ModeBit3 := FALSE;
   STATUS[916].EXT.BIT19 := FALSE;
   STATUS[916].EXT.BIT20 := FALSE;
   STATUS[916].EXT.AlarmSuppressed := FALSE;
   STATUS[916].EXT.AlarmPresent := FALSE;
   STATUS[916].EXT.AlarmFailUnAck := FALSE;
   STATUS[916].Status := 0;
   STATUS[916].TimeStamp := 16#0000;
   STATUS[917].EXT.AlarmWarnUnAck := FALSE;
   STATUS[917].EXT.AckRequired := FALSE;
   STATUS[917].EXT.Maintanence := FALSE;
   STATUS[917].EXT.Operation := FALSE;
   STATUS[917].EXT.Forced := FALSE;
   STATUS[917].EXT.BIT29 := FALSE;
   STATUS[917].EXT.BIT30 := FALSE;
   STATUS[917].EXT.BIT31 := FALSE;
   STATUS[917].EXT.ModeBit1 := FALSE;
   STATUS[917].EXT.ModeBit2 := FALSE;
   STATUS[917].EXT.ModeBit3 := FALSE;
   STATUS[917].EXT.BIT19 := FALSE;
   STATUS[917].EXT.BIT20 := FALSE;
   STATUS[917].EXT.AlarmSuppressed := FALSE;
   STATUS[917].EXT.AlarmPresent := FALSE;
   STATUS[917].EXT.AlarmFailUnAck := FALSE;
   STATUS[917].Status := 0;
   STATUS[917].TimeStamp := 16#0000;
   STATUS[918].EXT.AlarmWarnUnAck := FALSE;
   STATUS[918].EXT.AckRequired := FALSE;
   STATUS[918].EXT.Maintanence := FALSE;
   STATUS[918].EXT.Operation := FALSE;
   STATUS[918].EXT.Forced := FALSE;
   STATUS[918].EXT.BIT29 := FALSE;
   STATUS[918].EXT.BIT30 := FALSE;
   STATUS[918].EXT.BIT31 := FALSE;
   STATUS[918].EXT.ModeBit1 := FALSE;
   STATUS[918].EXT.ModeBit2 := FALSE;
   STATUS[918].EXT.ModeBit3 := FALSE;
   STATUS[918].EXT.BIT19 := FALSE;
   STATUS[918].EXT.BIT20 := FALSE;
   STATUS[918].EXT.AlarmSuppressed := FALSE;
   STATUS[918].EXT.AlarmPresent := FALSE;
   STATUS[918].EXT.AlarmFailUnAck := FALSE;
   STATUS[918].Status := 0;
   STATUS[918].TimeStamp := 16#0000;
   STATUS[919].EXT.AlarmWarnUnAck := FALSE;
   STATUS[919].EXT.AckRequired := FALSE;
   STATUS[919].EXT.Maintanence := FALSE;
   STATUS[919].EXT.Operation := FALSE;
   STATUS[919].EXT.Forced := FALSE;
   STATUS[919].EXT.BIT29 := FALSE;
   STATUS[919].EXT.BIT30 := FALSE;
   STATUS[919].EXT.BIT31 := FALSE;
   STATUS[919].EXT.ModeBit1 := FALSE;
   STATUS[919].EXT.ModeBit2 := FALSE;
   STATUS[919].EXT.ModeBit3 := FALSE;
   STATUS[919].EXT.BIT19 := FALSE;
   STATUS[919].EXT.BIT20 := FALSE;
   STATUS[919].EXT.AlarmSuppressed := FALSE;
   STATUS[919].EXT.AlarmPresent := FALSE;
   STATUS[919].EXT.AlarmFailUnAck := FALSE;
   STATUS[919].Status := 0;
   STATUS[919].TimeStamp := 16#0000;
   STATUS[920].EXT.AlarmWarnUnAck := FALSE;
   STATUS[920].EXT.AckRequired := FALSE;
   STATUS[920].EXT.Maintanence := FALSE;
   STATUS[920].EXT.Operation := FALSE;
   STATUS[920].EXT.Forced := FALSE;
   STATUS[920].EXT.BIT29 := FALSE;
   STATUS[920].EXT.BIT30 := FALSE;
   STATUS[920].EXT.BIT31 := FALSE;
   STATUS[920].EXT.ModeBit1 := FALSE;
   STATUS[920].EXT.ModeBit2 := FALSE;
   STATUS[920].EXT.ModeBit3 := FALSE;
   STATUS[920].EXT.BIT19 := FALSE;
   STATUS[920].EXT.BIT20 := FALSE;
   STATUS[920].EXT.AlarmSuppressed := FALSE;
   STATUS[920].EXT.AlarmPresent := FALSE;
   STATUS[920].EXT.AlarmFailUnAck := FALSE;
   STATUS[920].Status := 0;
   STATUS[920].TimeStamp := 16#0000;
   STATUS[921].EXT.AlarmWarnUnAck := FALSE;
   STATUS[921].EXT.AckRequired := FALSE;
   STATUS[921].EXT.Maintanence := FALSE;
   STATUS[921].EXT.Operation := FALSE;
   STATUS[921].EXT.Forced := FALSE;
   STATUS[921].EXT.BIT29 := FALSE;
   STATUS[921].EXT.BIT30 := FALSE;
   STATUS[921].EXT.BIT31 := FALSE;
   STATUS[921].EXT.ModeBit1 := FALSE;
   STATUS[921].EXT.ModeBit2 := FALSE;
   STATUS[921].EXT.ModeBit3 := FALSE;
   STATUS[921].EXT.BIT19 := FALSE;
   STATUS[921].EXT.BIT20 := FALSE;
   STATUS[921].EXT.AlarmSuppressed := FALSE;
   STATUS[921].EXT.AlarmPresent := FALSE;
   STATUS[921].EXT.AlarmFailUnAck := FALSE;
   STATUS[921].Status := 0;
   STATUS[921].TimeStamp := 16#0000;
   STATUS[922].EXT.AlarmWarnUnAck := FALSE;
   STATUS[922].EXT.AckRequired := FALSE;
   STATUS[922].EXT.Maintanence := FALSE;
   STATUS[922].EXT.Operation := FALSE;
   STATUS[922].EXT.Forced := FALSE;
   STATUS[922].EXT.BIT29 := FALSE;
   STATUS[922].EXT.BIT30 := FALSE;
   STATUS[922].EXT.BIT31 := FALSE;
   STATUS[922].EXT.ModeBit1 := FALSE;
   STATUS[922].EXT.ModeBit2 := FALSE;
   STATUS[922].EXT.ModeBit3 := FALSE;
   STATUS[922].EXT.BIT19 := FALSE;
   STATUS[922].EXT.BIT20 := FALSE;
   STATUS[922].EXT.AlarmSuppressed := FALSE;
   STATUS[922].EXT.AlarmPresent := FALSE;
   STATUS[922].EXT.AlarmFailUnAck := FALSE;
   STATUS[922].Status := 0;
   STATUS[922].TimeStamp := 16#0000;
   STATUS[923].EXT.AlarmWarnUnAck := FALSE;
   STATUS[923].EXT.AckRequired := FALSE;
   STATUS[923].EXT.Maintanence := FALSE;
   STATUS[923].EXT.Operation := FALSE;
   STATUS[923].EXT.Forced := FALSE;
   STATUS[923].EXT.BIT29 := FALSE;
   STATUS[923].EXT.BIT30 := FALSE;
   STATUS[923].EXT.BIT31 := FALSE;
   STATUS[923].EXT.ModeBit1 := FALSE;
   STATUS[923].EXT.ModeBit2 := FALSE;
   STATUS[923].EXT.ModeBit3 := FALSE;
   STATUS[923].EXT.BIT19 := FALSE;
   STATUS[923].EXT.BIT20 := FALSE;
   STATUS[923].EXT.AlarmSuppressed := FALSE;
   STATUS[923].EXT.AlarmPresent := FALSE;
   STATUS[923].EXT.AlarmFailUnAck := FALSE;
   STATUS[923].Status := 0;
   STATUS[923].TimeStamp := 16#0000;
   STATUS[924].EXT.AlarmWarnUnAck := FALSE;
   STATUS[924].EXT.AckRequired := FALSE;
   STATUS[924].EXT.Maintanence := FALSE;
   STATUS[924].EXT.Operation := FALSE;
   STATUS[924].EXT.Forced := FALSE;
   STATUS[924].EXT.BIT29 := FALSE;
   STATUS[924].EXT.BIT30 := FALSE;
   STATUS[924].EXT.BIT31 := FALSE;
   STATUS[924].EXT.ModeBit1 := FALSE;
   STATUS[924].EXT.ModeBit2 := FALSE;
   STATUS[924].EXT.ModeBit3 := FALSE;
   STATUS[924].EXT.BIT19 := FALSE;
   STATUS[924].EXT.BIT20 := FALSE;
   STATUS[924].EXT.AlarmSuppressed := FALSE;
   STATUS[924].EXT.AlarmPresent := FALSE;
   STATUS[924].EXT.AlarmFailUnAck := FALSE;
   STATUS[924].Status := 0;
   STATUS[924].TimeStamp := 16#0000;
   STATUS[925].EXT.AlarmWarnUnAck := FALSE;
   STATUS[925].EXT.AckRequired := FALSE;
   STATUS[925].EXT.Maintanence := FALSE;
   STATUS[925].EXT.Operation := FALSE;
   STATUS[925].EXT.Forced := FALSE;
   STATUS[925].EXT.BIT29 := FALSE;
   STATUS[925].EXT.BIT30 := FALSE;
   STATUS[925].EXT.BIT31 := FALSE;
   STATUS[925].EXT.ModeBit1 := FALSE;
   STATUS[925].EXT.ModeBit2 := FALSE;
   STATUS[925].EXT.ModeBit3 := FALSE;
   STATUS[925].EXT.BIT19 := FALSE;
   STATUS[925].EXT.BIT20 := FALSE;
   STATUS[925].EXT.AlarmSuppressed := FALSE;
   STATUS[925].EXT.AlarmPresent := FALSE;
   STATUS[925].EXT.AlarmFailUnAck := FALSE;
   STATUS[925].Status := 0;
   STATUS[925].TimeStamp := 16#0000;
   STATUS[926].EXT.AlarmWarnUnAck := FALSE;
   STATUS[926].EXT.AckRequired := FALSE;
   STATUS[926].EXT.Maintanence := FALSE;
   STATUS[926].EXT.Operation := FALSE;
   STATUS[926].EXT.Forced := FALSE;
   STATUS[926].EXT.BIT29 := FALSE;
   STATUS[926].EXT.BIT30 := FALSE;
   STATUS[926].EXT.BIT31 := FALSE;
   STATUS[926].EXT.ModeBit1 := FALSE;
   STATUS[926].EXT.ModeBit2 := FALSE;
   STATUS[926].EXT.ModeBit3 := FALSE;
   STATUS[926].EXT.BIT19 := FALSE;
   STATUS[926].EXT.BIT20 := FALSE;
   STATUS[926].EXT.AlarmSuppressed := FALSE;
   STATUS[926].EXT.AlarmPresent := FALSE;
   STATUS[926].EXT.AlarmFailUnAck := FALSE;
   STATUS[926].Status := 0;
   STATUS[926].TimeStamp := 16#0000;
   STATUS[927].EXT.AlarmWarnUnAck := FALSE;
   STATUS[927].EXT.AckRequired := FALSE;
   STATUS[927].EXT.Maintanence := FALSE;
   STATUS[927].EXT.Operation := FALSE;
   STATUS[927].EXT.Forced := FALSE;
   STATUS[927].EXT.BIT29 := FALSE;
   STATUS[927].EXT.BIT30 := FALSE;
   STATUS[927].EXT.BIT31 := FALSE;
   STATUS[927].EXT.ModeBit1 := FALSE;
   STATUS[927].EXT.ModeBit2 := FALSE;
   STATUS[927].EXT.ModeBit3 := FALSE;
   STATUS[927].EXT.BIT19 := FALSE;
   STATUS[927].EXT.BIT20 := FALSE;
   STATUS[927].EXT.AlarmSuppressed := FALSE;
   STATUS[927].EXT.AlarmPresent := FALSE;
   STATUS[927].EXT.AlarmFailUnAck := FALSE;
   STATUS[927].Status := 0;
   STATUS[927].TimeStamp := 16#0000;
   STATUS[928].EXT.AlarmWarnUnAck := FALSE;
   STATUS[928].EXT.AckRequired := FALSE;
   STATUS[928].EXT.Maintanence := FALSE;
   STATUS[928].EXT.Operation := FALSE;
   STATUS[928].EXT.Forced := FALSE;
   STATUS[928].EXT.BIT29 := FALSE;
   STATUS[928].EXT.BIT30 := FALSE;
   STATUS[928].EXT.BIT31 := FALSE;
   STATUS[928].EXT.ModeBit1 := FALSE;
   STATUS[928].EXT.ModeBit2 := FALSE;
   STATUS[928].EXT.ModeBit3 := FALSE;
   STATUS[928].EXT.BIT19 := FALSE;
   STATUS[928].EXT.BIT20 := FALSE;
   STATUS[928].EXT.AlarmSuppressed := FALSE;
   STATUS[928].EXT.AlarmPresent := FALSE;
   STATUS[928].EXT.AlarmFailUnAck := FALSE;
   STATUS[928].Status := 0;
   STATUS[928].TimeStamp := 16#0000;
   STATUS[929].EXT.AlarmWarnUnAck := FALSE;
   STATUS[929].EXT.AckRequired := FALSE;
   STATUS[929].EXT.Maintanence := FALSE;
   STATUS[929].EXT.Operation := FALSE;
   STATUS[929].EXT.Forced := FALSE;
   STATUS[929].EXT.BIT29 := FALSE;
   STATUS[929].EXT.BIT30 := FALSE;
   STATUS[929].EXT.BIT31 := FALSE;
   STATUS[929].EXT.ModeBit1 := FALSE;
   STATUS[929].EXT.ModeBit2 := FALSE;
   STATUS[929].EXT.ModeBit3 := FALSE;
   STATUS[929].EXT.BIT19 := FALSE;
   STATUS[929].EXT.BIT20 := FALSE;
   STATUS[929].EXT.AlarmSuppressed := FALSE;
   STATUS[929].EXT.AlarmPresent := FALSE;
   STATUS[929].EXT.AlarmFailUnAck := FALSE;
   STATUS[929].Status := 0;
   STATUS[929].TimeStamp := 16#0000;
   STATUS[930].EXT.AlarmWarnUnAck := FALSE;
   STATUS[930].EXT.AckRequired := FALSE;
   STATUS[930].EXT.Maintanence := FALSE;
   STATUS[930].EXT.Operation := FALSE;
   STATUS[930].EXT.Forced := FALSE;
   STATUS[930].EXT.BIT29 := FALSE;
   STATUS[930].EXT.BIT30 := FALSE;
   STATUS[930].EXT.BIT31 := FALSE;
   STATUS[930].EXT.ModeBit1 := FALSE;
   STATUS[930].EXT.ModeBit2 := FALSE;
   STATUS[930].EXT.ModeBit3 := FALSE;
   STATUS[930].EXT.BIT19 := FALSE;
   STATUS[930].EXT.BIT20 := FALSE;
   STATUS[930].EXT.AlarmSuppressed := FALSE;
   STATUS[930].EXT.AlarmPresent := FALSE;
   STATUS[930].EXT.AlarmFailUnAck := FALSE;
   STATUS[930].Status := 0;
   STATUS[930].TimeStamp := 16#0000;
   STATUS[931].EXT.AlarmWarnUnAck := FALSE;
   STATUS[931].EXT.AckRequired := FALSE;
   STATUS[931].EXT.Maintanence := FALSE;
   STATUS[931].EXT.Operation := FALSE;
   STATUS[931].EXT.Forced := FALSE;
   STATUS[931].EXT.BIT29 := FALSE;
   STATUS[931].EXT.BIT30 := FALSE;
   STATUS[931].EXT.BIT31 := FALSE;
   STATUS[931].EXT.ModeBit1 := FALSE;
   STATUS[931].EXT.ModeBit2 := FALSE;
   STATUS[931].EXT.ModeBit3 := FALSE;
   STATUS[931].EXT.BIT19 := FALSE;
   STATUS[931].EXT.BIT20 := FALSE;
   STATUS[931].EXT.AlarmSuppressed := FALSE;
   STATUS[931].EXT.AlarmPresent := FALSE;
   STATUS[931].EXT.AlarmFailUnAck := FALSE;
   STATUS[931].Status := 0;
   STATUS[931].TimeStamp := 16#0000;
   STATUS[932].EXT.AlarmWarnUnAck := FALSE;
   STATUS[932].EXT.AckRequired := FALSE;
   STATUS[932].EXT.Maintanence := FALSE;
   STATUS[932].EXT.Operation := FALSE;
   STATUS[932].EXT.Forced := FALSE;
   STATUS[932].EXT.BIT29 := FALSE;
   STATUS[932].EXT.BIT30 := FALSE;
   STATUS[932].EXT.BIT31 := FALSE;
   STATUS[932].EXT.ModeBit1 := FALSE;
   STATUS[932].EXT.ModeBit2 := FALSE;
   STATUS[932].EXT.ModeBit3 := FALSE;
   STATUS[932].EXT.BIT19 := FALSE;
   STATUS[932].EXT.BIT20 := FALSE;
   STATUS[932].EXT.AlarmSuppressed := FALSE;
   STATUS[932].EXT.AlarmPresent := FALSE;
   STATUS[932].EXT.AlarmFailUnAck := FALSE;
   STATUS[932].Status := 0;
   STATUS[932].TimeStamp := 16#0000;
   STATUS[933].EXT.AlarmWarnUnAck := FALSE;
   STATUS[933].EXT.AckRequired := FALSE;
   STATUS[933].EXT.Maintanence := FALSE;
   STATUS[933].EXT.Operation := FALSE;
   STATUS[933].EXT.Forced := FALSE;
   STATUS[933].EXT.BIT29 := FALSE;
   STATUS[933].EXT.BIT30 := FALSE;
   STATUS[933].EXT.BIT31 := FALSE;
   STATUS[933].EXT.ModeBit1 := FALSE;
   STATUS[933].EXT.ModeBit2 := FALSE;
   STATUS[933].EXT.ModeBit3 := FALSE;
   STATUS[933].EXT.BIT19 := FALSE;
   STATUS[933].EXT.BIT20 := FALSE;
   STATUS[933].EXT.AlarmSuppressed := FALSE;
   STATUS[933].EXT.AlarmPresent := FALSE;
   STATUS[933].EXT.AlarmFailUnAck := FALSE;
   STATUS[933].Status := 0;
   STATUS[933].TimeStamp := 16#0000;
   STATUS[934].EXT.AlarmWarnUnAck := FALSE;
   STATUS[934].EXT.AckRequired := FALSE;
   STATUS[934].EXT.Maintanence := FALSE;
   STATUS[934].EXT.Operation := FALSE;
   STATUS[934].EXT.Forced := FALSE;
   STATUS[934].EXT.BIT29 := FALSE;
   STATUS[934].EXT.BIT30 := FALSE;
   STATUS[934].EXT.BIT31 := FALSE;
   STATUS[934].EXT.ModeBit1 := FALSE;
   STATUS[934].EXT.ModeBit2 := FALSE;
   STATUS[934].EXT.ModeBit3 := FALSE;
   STATUS[934].EXT.BIT19 := FALSE;
   STATUS[934].EXT.BIT20 := FALSE;
   STATUS[934].EXT.AlarmSuppressed := FALSE;
   STATUS[934].EXT.AlarmPresent := FALSE;
   STATUS[934].EXT.AlarmFailUnAck := FALSE;
   STATUS[934].Status := 0;
   STATUS[934].TimeStamp := 16#0000;
   STATUS[935].EXT.AlarmWarnUnAck := FALSE;
   STATUS[935].EXT.AckRequired := FALSE;
   STATUS[935].EXT.Maintanence := FALSE;
   STATUS[935].EXT.Operation := FALSE;
   STATUS[935].EXT.Forced := FALSE;
   STATUS[935].EXT.BIT29 := FALSE;
   STATUS[935].EXT.BIT30 := FALSE;
   STATUS[935].EXT.BIT31 := FALSE;
   STATUS[935].EXT.ModeBit1 := FALSE;
   STATUS[935].EXT.ModeBit2 := FALSE;
   STATUS[935].EXT.ModeBit3 := FALSE;
   STATUS[935].EXT.BIT19 := FALSE;
   STATUS[935].EXT.BIT20 := FALSE;
   STATUS[935].EXT.AlarmSuppressed := FALSE;
   STATUS[935].EXT.AlarmPresent := FALSE;
   STATUS[935].EXT.AlarmFailUnAck := FALSE;
   STATUS[935].Status := 0;
   STATUS[935].TimeStamp := 16#0000;
   STATUS[936].EXT.AlarmWarnUnAck := FALSE;
   STATUS[936].EXT.AckRequired := FALSE;
   STATUS[936].EXT.Maintanence := FALSE;
   STATUS[936].EXT.Operation := FALSE;
   STATUS[936].EXT.Forced := FALSE;
   STATUS[936].EXT.BIT29 := FALSE;
   STATUS[936].EXT.BIT30 := FALSE;
   STATUS[936].EXT.BIT31 := FALSE;
   STATUS[936].EXT.ModeBit1 := FALSE;
   STATUS[936].EXT.ModeBit2 := FALSE;
   STATUS[936].EXT.ModeBit3 := FALSE;
   STATUS[936].EXT.BIT19 := FALSE;
   STATUS[936].EXT.BIT20 := FALSE;
   STATUS[936].EXT.AlarmSuppressed := FALSE;
   STATUS[936].EXT.AlarmPresent := FALSE;
   STATUS[936].EXT.AlarmFailUnAck := FALSE;
   STATUS[936].Status := 0;
   STATUS[936].TimeStamp := 16#0000;
   STATUS[937].EXT.AlarmWarnUnAck := FALSE;
   STATUS[937].EXT.AckRequired := FALSE;
   STATUS[937].EXT.Maintanence := FALSE;
   STATUS[937].EXT.Operation := FALSE;
   STATUS[937].EXT.Forced := FALSE;
   STATUS[937].EXT.BIT29 := FALSE;
   STATUS[937].EXT.BIT30 := FALSE;
   STATUS[937].EXT.BIT31 := FALSE;
   STATUS[937].EXT.ModeBit1 := FALSE;
   STATUS[937].EXT.ModeBit2 := FALSE;
   STATUS[937].EXT.ModeBit3 := FALSE;
   STATUS[937].EXT.BIT19 := FALSE;
   STATUS[937].EXT.BIT20 := FALSE;
   STATUS[937].EXT.AlarmSuppressed := FALSE;
   STATUS[937].EXT.AlarmPresent := FALSE;
   STATUS[937].EXT.AlarmFailUnAck := FALSE;
   STATUS[937].Status := 0;
   STATUS[937].TimeStamp := 16#0000;
   STATUS[938].EXT.AlarmWarnUnAck := FALSE;
   STATUS[938].EXT.AckRequired := FALSE;
   STATUS[938].EXT.Maintanence := FALSE;
   STATUS[938].EXT.Operation := FALSE;
   STATUS[938].EXT.Forced := FALSE;
   STATUS[938].EXT.BIT29 := FALSE;
   STATUS[938].EXT.BIT30 := FALSE;
   STATUS[938].EXT.BIT31 := FALSE;
   STATUS[938].EXT.ModeBit1 := FALSE;
   STATUS[938].EXT.ModeBit2 := FALSE;
   STATUS[938].EXT.ModeBit3 := FALSE;
   STATUS[938].EXT.BIT19 := FALSE;
   STATUS[938].EXT.BIT20 := FALSE;
   STATUS[938].EXT.AlarmSuppressed := FALSE;
   STATUS[938].EXT.AlarmPresent := FALSE;
   STATUS[938].EXT.AlarmFailUnAck := FALSE;
   STATUS[938].Status := 0;
   STATUS[938].TimeStamp := 16#0000;
   STATUS[939].EXT.AlarmWarnUnAck := FALSE;
   STATUS[939].EXT.AckRequired := FALSE;
   STATUS[939].EXT.Maintanence := FALSE;
   STATUS[939].EXT.Operation := FALSE;
   STATUS[939].EXT.Forced := FALSE;
   STATUS[939].EXT.BIT29 := FALSE;
   STATUS[939].EXT.BIT30 := FALSE;
   STATUS[939].EXT.BIT31 := FALSE;
   STATUS[939].EXT.ModeBit1 := FALSE;
   STATUS[939].EXT.ModeBit2 := FALSE;
   STATUS[939].EXT.ModeBit3 := FALSE;
   STATUS[939].EXT.BIT19 := FALSE;
   STATUS[939].EXT.BIT20 := FALSE;
   STATUS[939].EXT.AlarmSuppressed := FALSE;
   STATUS[939].EXT.AlarmPresent := FALSE;
   STATUS[939].EXT.AlarmFailUnAck := FALSE;
   STATUS[939].Status := 0;
   STATUS[939].TimeStamp := 16#0000;
   STATUS[940].EXT.AlarmWarnUnAck := FALSE;
   STATUS[940].EXT.AckRequired := FALSE;
   STATUS[940].EXT.Maintanence := FALSE;
   STATUS[940].EXT.Operation := FALSE;
   STATUS[940].EXT.Forced := FALSE;
   STATUS[940].EXT.BIT29 := FALSE;
   STATUS[940].EXT.BIT30 := FALSE;
   STATUS[940].EXT.BIT31 := FALSE;
   STATUS[940].EXT.ModeBit1 := FALSE;
   STATUS[940].EXT.ModeBit2 := FALSE;
   STATUS[940].EXT.ModeBit3 := FALSE;
   STATUS[940].EXT.BIT19 := FALSE;
   STATUS[940].EXT.BIT20 := FALSE;
   STATUS[940].EXT.AlarmSuppressed := FALSE;
   STATUS[940].EXT.AlarmPresent := FALSE;
   STATUS[940].EXT.AlarmFailUnAck := FALSE;
   STATUS[940].Status := 0;
   STATUS[940].TimeStamp := 16#0000;
   STATUS[941].EXT.AlarmWarnUnAck := FALSE;
   STATUS[941].EXT.AckRequired := FALSE;
   STATUS[941].EXT.Maintanence := FALSE;
   STATUS[941].EXT.Operation := FALSE;
   STATUS[941].EXT.Forced := FALSE;
   STATUS[941].EXT.BIT29 := FALSE;
   STATUS[941].EXT.BIT30 := FALSE;
   STATUS[941].EXT.BIT31 := FALSE;
   STATUS[941].EXT.ModeBit1 := FALSE;
   STATUS[941].EXT.ModeBit2 := FALSE;
   STATUS[941].EXT.ModeBit3 := FALSE;
   STATUS[941].EXT.BIT19 := FALSE;
   STATUS[941].EXT.BIT20 := FALSE;
   STATUS[941].EXT.AlarmSuppressed := FALSE;
   STATUS[941].EXT.AlarmPresent := FALSE;
   STATUS[941].EXT.AlarmFailUnAck := FALSE;
   STATUS[941].Status := 0;
   STATUS[941].TimeStamp := 16#0000;
   STATUS[942].EXT.AlarmWarnUnAck := FALSE;
   STATUS[942].EXT.AckRequired := FALSE;
   STATUS[942].EXT.Maintanence := FALSE;
   STATUS[942].EXT.Operation := FALSE;
   STATUS[942].EXT.Forced := FALSE;
   STATUS[942].EXT.BIT29 := FALSE;
   STATUS[942].EXT.BIT30 := FALSE;
   STATUS[942].EXT.BIT31 := FALSE;
   STATUS[942].EXT.ModeBit1 := FALSE;
   STATUS[942].EXT.ModeBit2 := FALSE;
   STATUS[942].EXT.ModeBit3 := FALSE;
   STATUS[942].EXT.BIT19 := FALSE;
   STATUS[942].EXT.BIT20 := FALSE;
   STATUS[942].EXT.AlarmSuppressed := FALSE;
   STATUS[942].EXT.AlarmPresent := FALSE;
   STATUS[942].EXT.AlarmFailUnAck := FALSE;
   STATUS[942].Status := 0;
   STATUS[942].TimeStamp := 16#0000;
   STATUS[943].EXT.AlarmWarnUnAck := FALSE;
   STATUS[943].EXT.AckRequired := FALSE;
   STATUS[943].EXT.Maintanence := FALSE;
   STATUS[943].EXT.Operation := FALSE;
   STATUS[943].EXT.Forced := FALSE;
   STATUS[943].EXT.BIT29 := FALSE;
   STATUS[943].EXT.BIT30 := FALSE;
   STATUS[943].EXT.BIT31 := FALSE;
   STATUS[943].EXT.ModeBit1 := FALSE;
   STATUS[943].EXT.ModeBit2 := FALSE;
   STATUS[943].EXT.ModeBit3 := FALSE;
   STATUS[943].EXT.BIT19 := FALSE;
   STATUS[943].EXT.BIT20 := FALSE;
   STATUS[943].EXT.AlarmSuppressed := FALSE;
   STATUS[943].EXT.AlarmPresent := FALSE;
   STATUS[943].EXT.AlarmFailUnAck := FALSE;
   STATUS[943].Status := 0;
   STATUS[943].TimeStamp := 16#0000;
   STATUS[944].EXT.AlarmWarnUnAck := FALSE;
   STATUS[944].EXT.AckRequired := FALSE;
   STATUS[944].EXT.Maintanence := FALSE;
   STATUS[944].EXT.Operation := FALSE;
   STATUS[944].EXT.Forced := FALSE;
   STATUS[944].EXT.BIT29 := FALSE;
   STATUS[944].EXT.BIT30 := FALSE;
   STATUS[944].EXT.BIT31 := FALSE;
   STATUS[944].EXT.ModeBit1 := FALSE;
   STATUS[944].EXT.ModeBit2 := FALSE;
   STATUS[944].EXT.ModeBit3 := FALSE;
   STATUS[944].EXT.BIT19 := FALSE;
   STATUS[944].EXT.BIT20 := FALSE;
   STATUS[944].EXT.AlarmSuppressed := FALSE;
   STATUS[944].EXT.AlarmPresent := FALSE;
   STATUS[944].EXT.AlarmFailUnAck := FALSE;
   STATUS[944].Status := 0;
   STATUS[944].TimeStamp := 16#0000;
   STATUS[945].EXT.AlarmWarnUnAck := FALSE;
   STATUS[945].EXT.AckRequired := FALSE;
   STATUS[945].EXT.Maintanence := FALSE;
   STATUS[945].EXT.Operation := FALSE;
   STATUS[945].EXT.Forced := FALSE;
   STATUS[945].EXT.BIT29 := FALSE;
   STATUS[945].EXT.BIT30 := FALSE;
   STATUS[945].EXT.BIT31 := FALSE;
   STATUS[945].EXT.ModeBit1 := FALSE;
   STATUS[945].EXT.ModeBit2 := FALSE;
   STATUS[945].EXT.ModeBit3 := FALSE;
   STATUS[945].EXT.BIT19 := FALSE;
   STATUS[945].EXT.BIT20 := FALSE;
   STATUS[945].EXT.AlarmSuppressed := FALSE;
   STATUS[945].EXT.AlarmPresent := FALSE;
   STATUS[945].EXT.AlarmFailUnAck := FALSE;
   STATUS[945].Status := 0;
   STATUS[945].TimeStamp := 16#0000;
   STATUS[946].EXT.AlarmWarnUnAck := FALSE;
   STATUS[946].EXT.AckRequired := FALSE;
   STATUS[946].EXT.Maintanence := FALSE;
   STATUS[946].EXT.Operation := FALSE;
   STATUS[946].EXT.Forced := FALSE;
   STATUS[946].EXT.BIT29 := FALSE;
   STATUS[946].EXT.BIT30 := FALSE;
   STATUS[946].EXT.BIT31 := FALSE;
   STATUS[946].EXT.ModeBit1 := FALSE;
   STATUS[946].EXT.ModeBit2 := FALSE;
   STATUS[946].EXT.ModeBit3 := FALSE;
   STATUS[946].EXT.BIT19 := FALSE;
   STATUS[946].EXT.BIT20 := FALSE;
   STATUS[946].EXT.AlarmSuppressed := FALSE;
   STATUS[946].EXT.AlarmPresent := FALSE;
   STATUS[946].EXT.AlarmFailUnAck := FALSE;
   STATUS[946].Status := 0;
   STATUS[946].TimeStamp := 16#0000;
   STATUS[947].EXT.AlarmWarnUnAck := FALSE;
   STATUS[947].EXT.AckRequired := FALSE;
   STATUS[947].EXT.Maintanence := FALSE;
   STATUS[947].EXT.Operation := FALSE;
   STATUS[947].EXT.Forced := FALSE;
   STATUS[947].EXT.BIT29 := FALSE;
   STATUS[947].EXT.BIT30 := FALSE;
   STATUS[947].EXT.BIT31 := FALSE;
   STATUS[947].EXT.ModeBit1 := FALSE;
   STATUS[947].EXT.ModeBit2 := FALSE;
   STATUS[947].EXT.ModeBit3 := FALSE;
   STATUS[947].EXT.BIT19 := FALSE;
   STATUS[947].EXT.BIT20 := FALSE;
   STATUS[947].EXT.AlarmSuppressed := FALSE;
   STATUS[947].EXT.AlarmPresent := FALSE;
   STATUS[947].EXT.AlarmFailUnAck := FALSE;
   STATUS[947].Status := 0;
   STATUS[947].TimeStamp := 16#0000;
   STATUS[948].EXT.AlarmWarnUnAck := FALSE;
   STATUS[948].EXT.AckRequired := FALSE;
   STATUS[948].EXT.Maintanence := FALSE;
   STATUS[948].EXT.Operation := FALSE;
   STATUS[948].EXT.Forced := FALSE;
   STATUS[948].EXT.BIT29 := FALSE;
   STATUS[948].EXT.BIT30 := FALSE;
   STATUS[948].EXT.BIT31 := FALSE;
   STATUS[948].EXT.ModeBit1 := FALSE;
   STATUS[948].EXT.ModeBit2 := FALSE;
   STATUS[948].EXT.ModeBit3 := FALSE;
   STATUS[948].EXT.BIT19 := FALSE;
   STATUS[948].EXT.BIT20 := FALSE;
   STATUS[948].EXT.AlarmSuppressed := FALSE;
   STATUS[948].EXT.AlarmPresent := FALSE;
   STATUS[948].EXT.AlarmFailUnAck := FALSE;
   STATUS[948].Status := 0;
   STATUS[948].TimeStamp := 16#0000;
   STATUS[949].EXT.AlarmWarnUnAck := FALSE;
   STATUS[949].EXT.AckRequired := FALSE;
   STATUS[949].EXT.Maintanence := FALSE;
   STATUS[949].EXT.Operation := FALSE;
   STATUS[949].EXT.Forced := FALSE;
   STATUS[949].EXT.BIT29 := FALSE;
   STATUS[949].EXT.BIT30 := FALSE;
   STATUS[949].EXT.BIT31 := FALSE;
   STATUS[949].EXT.ModeBit1 := FALSE;
   STATUS[949].EXT.ModeBit2 := FALSE;
   STATUS[949].EXT.ModeBit3 := FALSE;
   STATUS[949].EXT.BIT19 := FALSE;
   STATUS[949].EXT.BIT20 := FALSE;
   STATUS[949].EXT.AlarmSuppressed := FALSE;
   STATUS[949].EXT.AlarmPresent := FALSE;
   STATUS[949].EXT.AlarmFailUnAck := FALSE;
   STATUS[949].Status := 0;
   STATUS[949].TimeStamp := 16#0000;
   STATUS[950].EXT.AlarmWarnUnAck := FALSE;
   STATUS[950].EXT.AckRequired := FALSE;
   STATUS[950].EXT.Maintanence := FALSE;
   STATUS[950].EXT.Operation := FALSE;
   STATUS[950].EXT.Forced := FALSE;
   STATUS[950].EXT.BIT29 := FALSE;
   STATUS[950].EXT.BIT30 := FALSE;
   STATUS[950].EXT.BIT31 := FALSE;
   STATUS[950].EXT.ModeBit1 := FALSE;
   STATUS[950].EXT.ModeBit2 := FALSE;
   STATUS[950].EXT.ModeBit3 := FALSE;
   STATUS[950].EXT.BIT19 := FALSE;
   STATUS[950].EXT.BIT20 := FALSE;
   STATUS[950].EXT.AlarmSuppressed := FALSE;
   STATUS[950].EXT.AlarmPresent := FALSE;
   STATUS[950].EXT.AlarmFailUnAck := FALSE;
   STATUS[950].Status := 0;
   STATUS[950].TimeStamp := 16#0000;
   STATUS[951].EXT.AlarmWarnUnAck := FALSE;
   STATUS[951].EXT.AckRequired := FALSE;
   STATUS[951].EXT.Maintanence := FALSE;
   STATUS[951].EXT.Operation := FALSE;
   STATUS[951].EXT.Forced := FALSE;
   STATUS[951].EXT.BIT29 := FALSE;
   STATUS[951].EXT.BIT30 := FALSE;
   STATUS[951].EXT.BIT31 := FALSE;
   STATUS[951].EXT.ModeBit1 := FALSE;
   STATUS[951].EXT.ModeBit2 := FALSE;
   STATUS[951].EXT.ModeBit3 := FALSE;
   STATUS[951].EXT.BIT19 := FALSE;
   STATUS[951].EXT.BIT20 := FALSE;
   STATUS[951].EXT.AlarmSuppressed := FALSE;
   STATUS[951].EXT.AlarmPresent := FALSE;
   STATUS[951].EXT.AlarmFailUnAck := FALSE;
   STATUS[951].Status := 0;
   STATUS[951].TimeStamp := 16#0000;
   STATUS[952].EXT.AlarmWarnUnAck := FALSE;
   STATUS[952].EXT.AckRequired := FALSE;
   STATUS[952].EXT.Maintanence := FALSE;
   STATUS[952].EXT.Operation := FALSE;
   STATUS[952].EXT.Forced := FALSE;
   STATUS[952].EXT.BIT29 := FALSE;
   STATUS[952].EXT.BIT30 := FALSE;
   STATUS[952].EXT.BIT31 := FALSE;
   STATUS[952].EXT.ModeBit1 := FALSE;
   STATUS[952].EXT.ModeBit2 := FALSE;
   STATUS[952].EXT.ModeBit3 := FALSE;
   STATUS[952].EXT.BIT19 := FALSE;
   STATUS[952].EXT.BIT20 := FALSE;
   STATUS[952].EXT.AlarmSuppressed := FALSE;
   STATUS[952].EXT.AlarmPresent := FALSE;
   STATUS[952].EXT.AlarmFailUnAck := FALSE;
   STATUS[952].Status := 0;
   STATUS[952].TimeStamp := 16#0000;
   STATUS[953].EXT.AlarmWarnUnAck := FALSE;
   STATUS[953].EXT.AckRequired := FALSE;
   STATUS[953].EXT.Maintanence := FALSE;
   STATUS[953].EXT.Operation := FALSE;
   STATUS[953].EXT.Forced := FALSE;
   STATUS[953].EXT.BIT29 := FALSE;
   STATUS[953].EXT.BIT30 := FALSE;
   STATUS[953].EXT.BIT31 := FALSE;
   STATUS[953].EXT.ModeBit1 := FALSE;
   STATUS[953].EXT.ModeBit2 := FALSE;
   STATUS[953].EXT.ModeBit3 := FALSE;
   STATUS[953].EXT.BIT19 := FALSE;
   STATUS[953].EXT.BIT20 := FALSE;
   STATUS[953].EXT.AlarmSuppressed := FALSE;
   STATUS[953].EXT.AlarmPresent := FALSE;
   STATUS[953].EXT.AlarmFailUnAck := FALSE;
   STATUS[953].Status := 0;
   STATUS[953].TimeStamp := 16#0000;
   STATUS[954].EXT.AlarmWarnUnAck := FALSE;
   STATUS[954].EXT.AckRequired := FALSE;
   STATUS[954].EXT.Maintanence := FALSE;
   STATUS[954].EXT.Operation := FALSE;
   STATUS[954].EXT.Forced := FALSE;
   STATUS[954].EXT.BIT29 := FALSE;
   STATUS[954].EXT.BIT30 := FALSE;
   STATUS[954].EXT.BIT31 := FALSE;
   STATUS[954].EXT.ModeBit1 := FALSE;
   STATUS[954].EXT.ModeBit2 := FALSE;
   STATUS[954].EXT.ModeBit3 := FALSE;
   STATUS[954].EXT.BIT19 := FALSE;
   STATUS[954].EXT.BIT20 := FALSE;
   STATUS[954].EXT.AlarmSuppressed := FALSE;
   STATUS[954].EXT.AlarmPresent := FALSE;
   STATUS[954].EXT.AlarmFailUnAck := FALSE;
   STATUS[954].Status := 0;
   STATUS[954].TimeStamp := 16#0000;
   STATUS[955].EXT.AlarmWarnUnAck := FALSE;
   STATUS[955].EXT.AckRequired := FALSE;
   STATUS[955].EXT.Maintanence := FALSE;
   STATUS[955].EXT.Operation := FALSE;
   STATUS[955].EXT.Forced := FALSE;
   STATUS[955].EXT.BIT29 := FALSE;
   STATUS[955].EXT.BIT30 := FALSE;
   STATUS[955].EXT.BIT31 := FALSE;
   STATUS[955].EXT.ModeBit1 := FALSE;
   STATUS[955].EXT.ModeBit2 := FALSE;
   STATUS[955].EXT.ModeBit3 := FALSE;
   STATUS[955].EXT.BIT19 := FALSE;
   STATUS[955].EXT.BIT20 := FALSE;
   STATUS[955].EXT.AlarmSuppressed := FALSE;
   STATUS[955].EXT.AlarmPresent := FALSE;
   STATUS[955].EXT.AlarmFailUnAck := FALSE;
   STATUS[955].Status := 0;
   STATUS[955].TimeStamp := 16#0000;
   STATUS[956].EXT.AlarmWarnUnAck := FALSE;
   STATUS[956].EXT.AckRequired := FALSE;
   STATUS[956].EXT.Maintanence := FALSE;
   STATUS[956].EXT.Operation := FALSE;
   STATUS[956].EXT.Forced := FALSE;
   STATUS[956].EXT.BIT29 := FALSE;
   STATUS[956].EXT.BIT30 := FALSE;
   STATUS[956].EXT.BIT31 := FALSE;
   STATUS[956].EXT.ModeBit1 := FALSE;
   STATUS[956].EXT.ModeBit2 := FALSE;
   STATUS[956].EXT.ModeBit3 := FALSE;
   STATUS[956].EXT.BIT19 := FALSE;
   STATUS[956].EXT.BIT20 := FALSE;
   STATUS[956].EXT.AlarmSuppressed := FALSE;
   STATUS[956].EXT.AlarmPresent := FALSE;
   STATUS[956].EXT.AlarmFailUnAck := FALSE;
   STATUS[956].Status := 0;
   STATUS[956].TimeStamp := 16#0000;
   STATUS[957].EXT.AlarmWarnUnAck := FALSE;
   STATUS[957].EXT.AckRequired := FALSE;
   STATUS[957].EXT.Maintanence := FALSE;
   STATUS[957].EXT.Operation := FALSE;
   STATUS[957].EXT.Forced := FALSE;
   STATUS[957].EXT.BIT29 := FALSE;
   STATUS[957].EXT.BIT30 := FALSE;
   STATUS[957].EXT.BIT31 := FALSE;
   STATUS[957].EXT.ModeBit1 := FALSE;
   STATUS[957].EXT.ModeBit2 := FALSE;
   STATUS[957].EXT.ModeBit3 := FALSE;
   STATUS[957].EXT.BIT19 := FALSE;
   STATUS[957].EXT.BIT20 := FALSE;
   STATUS[957].EXT.AlarmSuppressed := FALSE;
   STATUS[957].EXT.AlarmPresent := FALSE;
   STATUS[957].EXT.AlarmFailUnAck := FALSE;
   STATUS[957].Status := 0;
   STATUS[957].TimeStamp := 16#0000;
   STATUS[958].EXT.AlarmWarnUnAck := FALSE;
   STATUS[958].EXT.AckRequired := FALSE;
   STATUS[958].EXT.Maintanence := FALSE;
   STATUS[958].EXT.Operation := FALSE;
   STATUS[958].EXT.Forced := FALSE;
   STATUS[958].EXT.BIT29 := FALSE;
   STATUS[958].EXT.BIT30 := FALSE;
   STATUS[958].EXT.BIT31 := FALSE;
   STATUS[958].EXT.ModeBit1 := FALSE;
   STATUS[958].EXT.ModeBit2 := FALSE;
   STATUS[958].EXT.ModeBit3 := FALSE;
   STATUS[958].EXT.BIT19 := FALSE;
   STATUS[958].EXT.BIT20 := FALSE;
   STATUS[958].EXT.AlarmSuppressed := FALSE;
   STATUS[958].EXT.AlarmPresent := FALSE;
   STATUS[958].EXT.AlarmFailUnAck := FALSE;
   STATUS[958].Status := 0;
   STATUS[958].TimeStamp := 16#0000;
   STATUS[959].EXT.AlarmWarnUnAck := FALSE;
   STATUS[959].EXT.AckRequired := FALSE;
   STATUS[959].EXT.Maintanence := FALSE;
   STATUS[959].EXT.Operation := FALSE;
   STATUS[959].EXT.Forced := FALSE;
   STATUS[959].EXT.BIT29 := FALSE;
   STATUS[959].EXT.BIT30 := FALSE;
   STATUS[959].EXT.BIT31 := FALSE;
   STATUS[959].EXT.ModeBit1 := FALSE;
   STATUS[959].EXT.ModeBit2 := FALSE;
   STATUS[959].EXT.ModeBit3 := FALSE;
   STATUS[959].EXT.BIT19 := FALSE;
   STATUS[959].EXT.BIT20 := FALSE;
   STATUS[959].EXT.AlarmSuppressed := FALSE;
   STATUS[959].EXT.AlarmPresent := FALSE;
   STATUS[959].EXT.AlarmFailUnAck := FALSE;
   STATUS[959].Status := 0;
   STATUS[959].TimeStamp := 16#0000;
   STATUS[960].EXT.AlarmWarnUnAck := FALSE;
   STATUS[960].EXT.AckRequired := FALSE;
   STATUS[960].EXT.Maintanence := FALSE;
   STATUS[960].EXT.Operation := FALSE;
   STATUS[960].EXT.Forced := FALSE;
   STATUS[960].EXT.BIT29 := FALSE;
   STATUS[960].EXT.BIT30 := FALSE;
   STATUS[960].EXT.BIT31 := FALSE;
   STATUS[960].EXT.ModeBit1 := FALSE;
   STATUS[960].EXT.ModeBit2 := FALSE;
   STATUS[960].EXT.ModeBit3 := FALSE;
   STATUS[960].EXT.BIT19 := FALSE;
   STATUS[960].EXT.BIT20 := FALSE;
   STATUS[960].EXT.AlarmSuppressed := FALSE;
   STATUS[960].EXT.AlarmPresent := FALSE;
   STATUS[960].EXT.AlarmFailUnAck := FALSE;
   STATUS[960].Status := 0;
   STATUS[960].TimeStamp := 16#0000;
   STATUS[961].EXT.AlarmWarnUnAck := FALSE;
   STATUS[961].EXT.AckRequired := FALSE;
   STATUS[961].EXT.Maintanence := FALSE;
   STATUS[961].EXT.Operation := FALSE;
   STATUS[961].EXT.Forced := FALSE;
   STATUS[961].EXT.BIT29 := FALSE;
   STATUS[961].EXT.BIT30 := FALSE;
   STATUS[961].EXT.BIT31 := FALSE;
   STATUS[961].EXT.ModeBit1 := FALSE;
   STATUS[961].EXT.ModeBit2 := FALSE;
   STATUS[961].EXT.ModeBit3 := FALSE;
   STATUS[961].EXT.BIT19 := FALSE;
   STATUS[961].EXT.BIT20 := FALSE;
   STATUS[961].EXT.AlarmSuppressed := FALSE;
   STATUS[961].EXT.AlarmPresent := FALSE;
   STATUS[961].EXT.AlarmFailUnAck := FALSE;
   STATUS[961].Status := 0;
   STATUS[961].TimeStamp := 16#0000;
   STATUS[962].EXT.AlarmWarnUnAck := FALSE;
   STATUS[962].EXT.AckRequired := FALSE;
   STATUS[962].EXT.Maintanence := FALSE;
   STATUS[962].EXT.Operation := FALSE;
   STATUS[962].EXT.Forced := FALSE;
   STATUS[962].EXT.BIT29 := FALSE;
   STATUS[962].EXT.BIT30 := FALSE;
   STATUS[962].EXT.BIT31 := FALSE;
   STATUS[962].EXT.ModeBit1 := FALSE;
   STATUS[962].EXT.ModeBit2 := FALSE;
   STATUS[962].EXT.ModeBit3 := FALSE;
   STATUS[962].EXT.BIT19 := FALSE;
   STATUS[962].EXT.BIT20 := FALSE;
   STATUS[962].EXT.AlarmSuppressed := FALSE;
   STATUS[962].EXT.AlarmPresent := FALSE;
   STATUS[962].EXT.AlarmFailUnAck := FALSE;
   STATUS[962].Status := 0;
   STATUS[962].TimeStamp := 16#0000;
   STATUS[963].EXT.AlarmWarnUnAck := FALSE;
   STATUS[963].EXT.AckRequired := FALSE;
   STATUS[963].EXT.Maintanence := FALSE;
   STATUS[963].EXT.Operation := FALSE;
   STATUS[963].EXT.Forced := FALSE;
   STATUS[963].EXT.BIT29 := FALSE;
   STATUS[963].EXT.BIT30 := FALSE;
   STATUS[963].EXT.BIT31 := FALSE;
   STATUS[963].EXT.ModeBit1 := FALSE;
   STATUS[963].EXT.ModeBit2 := FALSE;
   STATUS[963].EXT.ModeBit3 := FALSE;
   STATUS[963].EXT.BIT19 := FALSE;
   STATUS[963].EXT.BIT20 := FALSE;
   STATUS[963].EXT.AlarmSuppressed := FALSE;
   STATUS[963].EXT.AlarmPresent := FALSE;
   STATUS[963].EXT.AlarmFailUnAck := FALSE;
   STATUS[963].Status := 0;
   STATUS[963].TimeStamp := 16#0000;
   STATUS[964].EXT.AlarmWarnUnAck := FALSE;
   STATUS[964].EXT.AckRequired := FALSE;
   STATUS[964].EXT.Maintanence := FALSE;
   STATUS[964].EXT.Operation := FALSE;
   STATUS[964].EXT.Forced := FALSE;
   STATUS[964].EXT.BIT29 := FALSE;
   STATUS[964].EXT.BIT30 := FALSE;
   STATUS[964].EXT.BIT31 := FALSE;
   STATUS[964].EXT.ModeBit1 := FALSE;
   STATUS[964].EXT.ModeBit2 := FALSE;
   STATUS[964].EXT.ModeBit3 := FALSE;
   STATUS[964].EXT.BIT19 := FALSE;
   STATUS[964].EXT.BIT20 := FALSE;
   STATUS[964].EXT.AlarmSuppressed := FALSE;
   STATUS[964].EXT.AlarmPresent := FALSE;
   STATUS[964].EXT.AlarmFailUnAck := FALSE;
   STATUS[964].Status := 0;
   STATUS[964].TimeStamp := 16#0000;
   STATUS[965].EXT.AlarmWarnUnAck := FALSE;
   STATUS[965].EXT.AckRequired := FALSE;
   STATUS[965].EXT.Maintanence := FALSE;
   STATUS[965].EXT.Operation := FALSE;
   STATUS[965].EXT.Forced := FALSE;
   STATUS[965].EXT.BIT29 := FALSE;
   STATUS[965].EXT.BIT30 := FALSE;
   STATUS[965].EXT.BIT31 := FALSE;
   STATUS[965].EXT.ModeBit1 := FALSE;
   STATUS[965].EXT.ModeBit2 := FALSE;
   STATUS[965].EXT.ModeBit3 := FALSE;
   STATUS[965].EXT.BIT19 := FALSE;
   STATUS[965].EXT.BIT20 := FALSE;
   STATUS[965].EXT.AlarmSuppressed := FALSE;
   STATUS[965].EXT.AlarmPresent := FALSE;
   STATUS[965].EXT.AlarmFailUnAck := FALSE;
   STATUS[965].Status := 0;
   STATUS[965].TimeStamp := 16#0000;
   STATUS[966].EXT.AlarmWarnUnAck := FALSE;
   STATUS[966].EXT.AckRequired := FALSE;
   STATUS[966].EXT.Maintanence := FALSE;
   STATUS[966].EXT.Operation := FALSE;
   STATUS[966].EXT.Forced := FALSE;
   STATUS[966].EXT.BIT29 := FALSE;
   STATUS[966].EXT.BIT30 := FALSE;
   STATUS[966].EXT.BIT31 := FALSE;
   STATUS[966].EXT.ModeBit1 := FALSE;
   STATUS[966].EXT.ModeBit2 := FALSE;
   STATUS[966].EXT.ModeBit3 := FALSE;
   STATUS[966].EXT.BIT19 := FALSE;
   STATUS[966].EXT.BIT20 := FALSE;
   STATUS[966].EXT.AlarmSuppressed := FALSE;
   STATUS[966].EXT.AlarmPresent := FALSE;
   STATUS[966].EXT.AlarmFailUnAck := FALSE;
   STATUS[966].Status := 0;
   STATUS[966].TimeStamp := 16#0000;
   STATUS[967].EXT.AlarmWarnUnAck := FALSE;
   STATUS[967].EXT.AckRequired := FALSE;
   STATUS[967].EXT.Maintanence := FALSE;
   STATUS[967].EXT.Operation := FALSE;
   STATUS[967].EXT.Forced := FALSE;
   STATUS[967].EXT.BIT29 := FALSE;
   STATUS[967].EXT.BIT30 := FALSE;
   STATUS[967].EXT.BIT31 := FALSE;
   STATUS[967].EXT.ModeBit1 := FALSE;
   STATUS[967].EXT.ModeBit2 := FALSE;
   STATUS[967].EXT.ModeBit3 := FALSE;
   STATUS[967].EXT.BIT19 := FALSE;
   STATUS[967].EXT.BIT20 := FALSE;
   STATUS[967].EXT.AlarmSuppressed := FALSE;
